	b_first_pos_done:BOOL;
	b_second_pos_done:BOOL;
	b_3rd_pos_done:BOOL;
	b_4th_pos_done:BOOL;
	b_5th_pos_done:BOOL;
	b_6th_pos_done:BOOL;
	b_7th_pos_done:BOOL;
	b_8th_pos_done:BOOL;
	b_9th_pos_done:BOOL;
	b_10th_pos_done:BOOL;
	i_adjust_count:INT:=0;
	adjust_delay:BOOL;
	i_closeloop_count:INT:=0;
	rSPEED: REAL:=2500;
	rACC:REAL:=100;
	rDCC:REAL:=100;
	r_vel_EL_temp:LREAL;
	add_vel:LREAL;
	r_vel_EL:LREAL;
	b_modify_vel: BOOL;
	b_start_adjust_vel:BOOL;
	b_start_adjust_vel_temp:BOOL;
	r_compensation_value_motor: LREAL;
	r_compensation_abs: LREAL;
	b_test_offset_start:BOOL;
	r_offset_az_old:LREAL;
	r_offset_el_old:LREAL;
(*EL  vel mode*)	
	V_LastOutput:LREAL:=0;
	V_LastSpeed:LREAL:=0;
	dIntegralSpeed:LREAL:= 0;	
	V_command_EL:LREAL:=0;
	V_command_EL_V:LREAL:=0;

	V_max_vel_motor:LREAL;
	b_start_cyclicvel: BOOL;
	b_write_el_vel: BOOL;
	m_dLastIntegral:LREAL:=0;
	m_dAUnsub1:LREAL:=0;
	m_dAUnsub2:LREAL:=0;
	m_dAEnsub1:LREAL:=0;
	m_dAEnsub2:LREAL:=0;
	m_dKa:LREAL:=0.5;
	m_dKv:LREAL:=0.1;
	
	speed1:LREAL;
	r_EL_current_when_goto_cmd:LREAL;
	T_count_goto:LREAL;
	Pos_EL_Aim:LREAL;
	r_cyclic_velocity:LREAL;
	r_cyclic_velocity_test:LREAL;
	Pos_EL_error:LREAL;
	b_step_running:BOOL:=0;
	b_step_running_az:BOOL:=0;
	b_step_running_el:BOOL:=0;
	r_step_count:DINT:=0;
	r_step_count_temp:DINT:=0;
	b_offset_running:BOOL;
	r_offset_count_temp:DINT:=0;
	r_offset_count:DINT:=0;
	r_test_offset_az:LREAL;
	r_test_offset_el:LREAL;
	r_Integral_thistime:REAL;
	r_el_offset_abs:LREAL;
END_VAR
VAR_GLOBAL RETAIN PERSISTENT
	AZ_encoder_last: LREAL;
	FI_encoder_last: LREAL;

(*	
	C1:REAL:=-0.504475;
	C2:REAL:=-0.047962;
	C3:REAL:=0.005718;
	C4:REAL:=50.64244;
	C5:REAL:=-0.003995;
	C6:REAL:=0.443004;
	C7:REAL:=0.019635;
	C8:REAL:=0;
*)	

(*	C1:LREAL:=0;
	C2:LREAL:=0;
	C3:LREAL:=0;
	C4:LREAL:=0;
	C5:LREAL:=0;
	C6:LREAL:=0;
	C7:LREAL:=0;
	C8:LREAL:=0;	
*)
	r_pos_motor3_Ini: REAL;

(*	
	P1:LREAL:=0.000000000968559949;
	P2:LREAL:=-0.000000404463748;
	P3:LREAL:=0.0000707747355;
	P4:LREAL:=-0.006745089;
	P5:LREAL:=0.3810258947;
	P6:LREAL:=-13.13945082;
	P7:LREAL:=311.5666046431;
	P8:LREAL:=4122.813236;
	P9:LREAL:=556099.6655657330;
*)
	P1:LREAL:=0.00000000000675664022381225;
	P2:LREAL:=-0.00000000306148315353895;
	P3:LREAL:=0.000000597917575287703;
	P4:LREAL:=-0.0000659096897179393;
	P5:LREAL:=0.00450794567760492;
	P6:LREAL:=-0.198139695223752;
	P7:LREAL:=5.43570049374671;
	P8:LREAL:=-35.3877608207139;
	P9:LREAL:=9702.49448593394;
	P10:LREAL:=422614.297996071;
	
	AA1:LREAL:=0.0000927334099929522;
	AA2:LREAL:=0.0000884282758254779;
	AA3:LREAL:=0.0000846410373605538;
	AA4:LREAL:=0.0000813259380946959;
	AA5:LREAL:=0.0000784067743453034;
	AA6:LREAL:=0.000075826508947528;
	AA7:LREAL:=0.0000735467168745587;
	AA8:LREAL:=0.0000715348517797871;
	AA9:LREAL:=0.0000697632236190369;
	AA10:LREAL:=0.0000682035193015959;
	AA11:LREAL:=0.0000668341977222905;
	AA12:LREAL:=0.0000656452269355495;
	AA13:LREAL:=0.0000646345562191369;
	AA14:LREAL:=0.0000637852732561106;
	AA15:LREAL:=0.000063021502936802;
	
	BB1:LREAL:=37.4712526429021;
	BB2:LREAL:=34.8032470862882;
	BB3:LREAL:=32.2419717976062;
	BB4:LREAL:=29.8041671410679;
	BB5:LREAL:=27.4781245099576;
	BB6:LREAL:=25.2575068243857;
	BB7:LREAL:=23.1452253471404;
	BB8:LREAL:=21.1443430239212;
	BB9:LREAL:=19.2586262226003;
	BB10:LREAL:=17.4866321102168;
	BB11:LREAL:=15.8306154092925;
	BB12:LREAL:=14.3037010778946;
	BB13:LREAL:=12.9288502805138;
	BB14:LREAL:=11.7078506914323;
	BB15:LREAL:=10.5498626131235;
	
END_VAR

// IndraMotionMlc1/Application/UserConstGlobal
VAR_GLOBAL CONSTANT
  // define all possible axis, set to maximum axis index to preserve ressources 
  // set to a maximum of 32 for the L45 and 16? for the L25
  uiMAX_AXIS_INDEX:   UINT    := INT_TO_UINT(MB_MAX_AXIS_NUMBER);
  
  // Simulation related
 	 gc_b_sim_on: BOOL :=0;  // True is simulation code activated. 
  // Azimuth limits
  	gc_r_limit_cw_az_sim:REAL:= 271 ;
	gc_r_limit_ccw_az_sim:REAL:= -271;
	gc_r_limit_final_cw_az_sim:REAL:= 271.2 ;
	gc_r_limit_final_ccw_az_sim:REAL:=-271.2 ;
 // Elevation Limits
	gc_r_limit_cw_el_sim:REAL:= 90.2;
	gc_r_limit_ccw_el_sim:REAL:= 14.8 ;
	gc_r_limit_final_cw_el_sim:REAL:=90.5 ;
	gc_r_limit_final_ccw_el_sim:REAL:=14.5 ;
 // Feed Indexer Limits
	gc_r_limit_cw_fi_sim:REAL:= 108;
	gc_r_limit_ccw_fi_sim:REAL:= -108;
	gc_r_limit_final_cw_fi_sim:REAL:= 108.2 ;
	gc_r_limit_final_ccw_fi_sim:REAL:= -108.2;
  
  // Time related 
  gc_UnixToSKAEpoch: LREAL := 946684768 ; //Seconds
  gc_SKAEpochMJD: LREAL := 51544; // MJD
  gc_KAPB_NTP: STRING :='10.97.64.1';
  gc_ITF_NTP: STRING:= '10.165.3.12 ';
  
 (* // Position limits
  gc_r_pos_max_Az: REAL := 271;
  gc_r_pos_min_Az: REAL := -271;  
  gc_r_pos_max_El: REAL := 90.2;
  gc_r_pos_min_El: REAL := 14.8;  
  gc_r_pos_max_Fi: REAL := 106;
  gc_r_pos_min_Fi: REAL := -106;  *)

   // Position limits
  gc_r_pos_max_Az: REAL := 271;
  gc_r_pos_min_Az: REAL := -271;  
  gc_r_pos_max_El: REAL := 90.20;
  gc_r_pos_min_El: REAL := -14.80;  
  gc_r_pos_max_Fi: REAL := 106;
  gc_r_pos_min_Fi: REAL := -106;  
  
  
  // Velocity limits
   gc_r_vel_max_Az: REAL := 0.5; //3/6; //scaling RPM of Axis  Deg/s = 6* RPM 
   gc_r_vel_max_El: REAL := 0.16667;
   gc_r_vel_max_Fi: REAL := 2;
   
  // Power limiting
     gc_r_power_Kv_Az: REAL := 0.05;//0.3Deg/s/kW;
  	 gc_r_power_Kv_El: REAL := 0.016667;// 0.1;
     gc_r_power_Kv_Fi: REAL := 0.2;//1.2;
	 gc_r_power_Ka_Az: REAL := 0.055;
  	 gc_r_power_Ka_El: REAL := 0.002;
  	 gc_r_power_Ka_Fi: REAL := 0.1; 

     
   // Tracking  If the velocity is below this limit then then the dish is tracking abovethe limit it is slewing. 
   gc_r_vel_tracking_limit_Az: REAL := 1;  // Scaling
   gc_r_vel_tracking_limit_El: REAL := 0.4;
   gc_r_vel_tracking_limit_Fi: REAL := 0;
   
   // Stop Deceleration values  
  gc_r_Stop_dec_Az: REAL := 0.5; //Rad/s^2
  gc_r_Stop_dec_El: REAL := 0.5; // 28,64 deg/s^2
  gc_r_Stop_dec_Fi: REAL := 0.5;
  
   // Stop Deceleration values  
  gc_r_limit_Stop_dec_Az: REAL := 5; //Rad/s^2
  gc_r_limit_Stop_dec_El: REAL := 5; // 28,64 deg/s^2
  gc_r_limit_Stop_dec_Fi: REAL := 5;
  
  
  // Goto Acceleration Values
  gc_r_goto_acc_Az: REAL := 0.02; //Rad/s^2 
  gc_r_goto_acc_El: REAL := 0.02; // 1.14 deg/s^@
  gc_r_goto_acc_Fi: REAL := 0.2; // 11.4 deg/s^2
  
  // Feed indexer positions for bands
  gc_r_band_tolerance: REAL := 0.001; // Tolerance for being in position
  gc_r_band_optical : REAL := 0;
  gc_r_band_1 : REAL := 103.37;
  gc_r_band_2 : REAL := -99.97;
  gc_r_band_3 : REAL := -47.684;
  gc_r_band_4 : REAL := 10.444;
  gc_r_band_5a : REAL := -6.398;
  gc_r_band_5b : REAL := -30.842;
  gc_r_band_6 : REAL := -18.62;
  
  // Stow Positions
  gc_r_stow_Az: REAL :=0; 
  gc_r_stow_El: REAL :=90;
  gc_stow_horn_alarm_time: TIME := T#5S;
  gc_UPS_Stow_Az_Speed: REAL := 0.16667;
  gc_UPS_Stow_El_Speed: REAL := 0.083; 
  // AutoStow 
  gc_i_autostow_counter_max: INT := 2; 
  
  // Static off set limits
  gc_r_Xel_off_limit: REAL := 36000; // arcsec
  gc_r_El_off_limit: REAL := 36000;
	 
  // Pointing 
  gc_stack_length: INT :=10000; 
  gc_r_tilt_vel_limit_Az: REAL := 1; // deg/s	 
  gc_lr_tilt_corr_limit_Az: LREAL:= 1000; //arcseconds 
  gc_lr_tilt_corr_limit_El: LREAL:= 1000; //arcseconds 
  gc_lr_arcsec2deg: LREAL:=3600;
  gc_lr_point_corr_error_lim : LREAL := 360000; //arcseconds
  
  // DAM 
  gc_st_DAM_ip:String :='192.168.1.222';
	 
END_VAR

// IndraMotionMlc1/Application/UserVarGlobal
VAR_GLOBAL 
  // Axis interface: command structure: define as RETAIN, to keep the values 
  // Note: on the L40.2 control, the RETAIN memory is slower then normal VAR, so define 
  //       this structure only as RETAIN when necessary 
  //  arAxisCtrl_gb: ARRAY [1..MAX_AXIS_NUM] OF MB_AXIS_CONTROL;
	
  // Axis interface: command structure 
  arAxisCtrl_gb: ARRAY [1..uiMAX_AXIS_INDEX] OF TE_AXIS_CONTROL_TYPE01;
END_VAR

VAR_GLOBAL
//----------------------------------- Machine status variables ----------------------------	

  // Axis interface: status structure 
  arAxisStatus_gb: ARRAY [1..uiMAX_AXIS_INDEX] OF TE_AXIS_STATUS_TYPE01;

  bRemoteOn_gb  : BOOL := FALSE;  // TRUE: Internal IL visu is active 
                                  // FALSE: PlcProg is active

  
END_VAR

// IndraMotionMlc1/Application/AxisInterface/Global_AxIf_Const
{attribute 'qualified_only'}
VAR_GLOBAL CONSTANT
    // define masks for the sync operating modes 
    // e.g. IF( (INT_TO_WORD(AdminStatus._OpMode.enAck) AND MASK_MODE_WITH_FINE_ADJ) <> 0 ) THEN 
    MASK_MODE_PHASE_SHIFT   :DWORD := 16#0BC0; (* SYNC_PHASE, SYNC_CAM, SYNC_PROFILE, FLEX_PROFILE, SYNC_VEL *)
END_VAR
VAR_GLOBAL

END_VAR

// IndraMotionMlc1/Application/AxisInterface/Global_Axis_Interface
{attribute 'linkalways'}
{attribute 'analysis' := '-33'} // disable static code analysis rule 33, check of unused variable
VAR_GLOBAL
    (* Axis number for the visualization screens *)
    VisuAxisNo : INT := 1;
    
	  arAxisIdx_gb: ARRAY [1..uiMAX_AXIS_INDEX] OF UINT; // list of all axes index without gaps 
    uiNofAxis_gb: UINT; // number of axis in C-0-0484
    
END_VAR

// IndraMotionMlc1/Application/PLC_PRG
VAR_GLOBAL
		
Safety:fb_Safety;
CommandArbiter:fb_CommandArbiter;
Time_cds:fb_Time_cds;
Pointing:fb_Pointing;
Tracking:fb_Tracking;
Management:fb_Management;
Azimuth:fb_Axis;
Elevation:fb_Axis;
FeedIndexer:fb_Axis;





	
(************CommandArbiter ************)	

	Authority:STRING:='LMC';    (* the authority for DSC control now*)
	Command_Arbiter_error:BOOL;(*Command Arbiter error*)

(****************Management*******************)

	DsState:UINT;(*The Dish state 0Startup 1Standby 2Locked 3Estop 4Stowed 5Lcok&Stowed 6Activating 7Deactivating 8Standstill 9Stop 10Slew 11jog 12Track*)
	Current_FIPos:UINT;(*Current position of the FI*)
	r_operation_hour: LREAL;(*FP_C_0_0051,Operation hour counter*)
	K_gear_ratio:LREAL:=1800;// The ratio beteen the leadscrew length and elevation angle This variable needs a non-zero startup to prevent divide by zero.
	HumidDriveCab: LREAL;
	HumidDriveCab_Up: LREAL;
	HumidPSC_Inlet: LREAL;
	HumidPSC_Outlet: LREAL;
	TempDriveCab: LREAL;
	TempDriveCab_Up: LREAL;
	TempEMISC_Outlet: LREAL;
	TempPSC_Inlet: LREAL;
	TempPSC_Outlet: LREAL;
	CurrentPh1: LREAL;
	CurrentPh2: LREAL;
	CurrentPh3: LREAL;
	FrequencyPh1: LREAL;
	FrequencyPh2: LREAL;
	FrequencyPh3: LREAL;
	PowerFactor: LREAL;
	VoltagePh1: LREAL;
	VoltagePh2: LREAL;
	VoltagePh3: LREAL;
	
	Pedestal_temp_1: REAL;
	Pedestal_temp_2 : REAL;
	Pedestal_temp_3 : REAL;
	
	ActivePowerConsumption: LREAL;
	ReactivePowerConsumption: LREAL;
	ApparentPowerConsumption: LREAL;
		
(********************Time**********************)	
	Source_Timesync:UINT:=2;(*Time source, 0 PTP 1 NTP 2 DSC*)
	IP_Adress_PTP:STRING;(* The PTP server adresss*)
	IP_Adress_NTP:STRING;(* The PTP server adresss*)
	//DscTime:DATE_AND_TIME;(*DSC internal time*)
	//TimeSynced:BOOL;(*The time is synced to the source*)
	
(**********************Pointing************************)	
	(*ActAmbTemp_East:LREAL;
	ActAmbTemp_South:LREAL;
	AmbTempCorrVal_1:LREAL;
	AmbTempCorrVal_2:LREAL;
	TiltXRaw_One:LREAL;
	TiltYRaw_One:LREAL;
	TiltXArcsec_One:LREAL;
	TiltYArcsec_One: BOOL;
	TiltXFilt_One:LREAL;
	TiltYFilt_One:LREAL;
	TiltTemp_One:LREAL;
	TiltXRaw_Two:LREAL;
	TiltYRaw_Two:LREAL;
	TiltXArcsec_Two:LREAL;
	TiltYArcsec_Two: BOOL;
	TiltXFilt_Two:LREAL;
	TiltYFilt_Two:LREAL;
	TiltTemp_Two:LREAL;
	TiltCorrVal_Az:LREAL;
	TiltCorrVal_EL:LREAL;
	PmCorrVal_Az: BOOL;
	PmCorrVal_EL: BOOL;
	StaticCorrActive:BOOL;
	TiltCorrActive:BOOL;
	Pointing_TiltOn:UINT;
	TempCorrActive:BOOL;
	BandForCorr:UINT;*)
	Pointing_TiltOn:UINT;
(**************************Tracking********************************)
(*	tr_initOk:BOOL;(*Tracking function program is initialized and ready for operation*)
	tr_valid:BOOL;(*The tracking controller’s output is within the position ranges of the dish structure.*)
	tr_Table_error:BOOL;(*The table reports an error *)
	tr_obj_valid:BOOL;(*Tracking object has valid tracking data.*)
	tr_selFIy:BOOL;(*FIynomial tracking selected as source*)
	act_statOffset_value_Xel:LREAL;(*Actual azimuth static offset*)
	act_statOffset_value_El:LREAL;(*Elevation azimuth static offset*)
	p_desired_AZ:LREAL;(*Azimuth position output of the Tracking Controller*)
	p_desired_EL:LREAL;(*Elevation position output of the Tracking Controller*)
	tr_TimeRemaining:LREAL;(*Time till the last point in the track table is reached*)
	OnSourceDev:LREAL;(*Actual calculated “On Sky” rms tracking error.*) *)
(*********Read parameteers*******)
	AxRef:ARRAY[1..5] OF AXIS_REF;
	P_shape_value:ARRAY[1..5] OF LREAL;
	V_shape_value:ARRAY[1..5] OF LREAL;
	V_act_value:ARRAY[1..5] OF LREAL;
	r_write_position_az: LREAL; // Used internally for interpolator and pointing model calculations
    r_write_position_az_out: LREAL; (*the position written to the virvual azimuth axis*)
	r_write_position_el: LREAL; // Used internally for interpolator and pointing model calculations
    r_write_position_el_out: LREAL;(*the position written to the virvual elevation axis*)
	r_write_position_FI: LREAL;(*the position written to the virvual FeedIndexer axis*)
	r_write_position_FI_out: LREAL;(*the position written to the virvual FeedIndexer axis*)
	
END_VAR

VAR_GLOBAL RETAIN PERSISTENT
	R_total_distance_AZ:LREAL;
	R_total_distance_EL_deg:LREAL;
	R_total_distance_EL_m:LREAL;
	R_total_distance_FI:LREAL;
	
	LeapSecPTP: UINT :=37;    // Storage for Leap seconds 
	
END_VAR

// IndraMotionMlc1/Application/POUs/Motion/P_Position_and_MJD
(*The program is built for calculating the position of real axis, virtual axis and the MJD time,
and writing software limit of azimuth *)
PROGRAM P_Position_and_MJD
VAR
(*With the function block "MB_WriteRealParameter" you can write a defined value to the parameter belonging to the parameter number*)
	fb_write_negative_a: MB_WriteRealParameter;
	fb_write_negative_s: MB_WriteRealParameter;
	fb_write_positive_a: MB_WriteRealParameter;
	fb_write_positive_s: MB_WriteRealParameter;
(*the blink function block is for triggering MB_WriteRealParameter function block*)
	fb_blink_1: BLINK;
	fb_blink_2: BLINK;
	fb_blink_3: BLINK;
	fb_blink_4: BLINK;
(*the value is written to MB_WriteRealParameter*)
	r_negative_limit: REAL;
	r_positive_limit: REAL;
(*the elevation limit control*)
	fb_blink_diagnos_el: BLINK;
	fb_diagnose_el: MB_ReadStringParameter;
	str_diagnose_el: STRING;
	fb_blink_5: BLINK;
	fb_blink_6: BLINK;
	fb_write_negative_el: MB_WriteRealParameter;
	fb_write_positive_el: MB_WriteRealParameter;
	r_limit_el_up: REAL;
	r_limit_el_down: REAL;
	b_limit_up_el: BOOL;
	b_limit_down_el: BOOL;
	rtrig_set_limit_up: R_TRIG;
	rtrig_set_limit_down: R_TRIG;
	fb_blink_7: BLINK;
	fb_write_91_az1: MB_WriteRealParameter;
	fb_blink_8: BLINK;
	fb_blink_9: BLINK;
	fb_blink_10: BLINK;
	fb_blink_11: BLINK;
	fb_write_91_az2: MB_WriteRealParameter;
	fb_write_91_el1: MB_WriteRealParameter;
	fb_write_91_el2: MB_WriteRealParameter;
	fb_write_91_FI: MB_WriteRealParameter;
	fb_blink_12: BLINK;
	fb_write_91_FI2: MB_WriteRealParameter;
	r_pos_FI_1: REAL;
	i_counter_hr: BOOL;
	rtrig_hr:R_TRIG;
	
	fb_blink_111: BLINK;
	fb_write_negative_a_v: MB_WriteRealParameter;
	fb_blink_1_v: BLINK;
	fb_blink_2_v: BLINK;
	fb_write_negative_s_v: MB_WriteRealParameter;
	fb_blink_3_v: BLINK;
	fb_write_positive_a_v: MB_WriteRealParameter;
	
	temp_a:LREAL:=3135.4451;
	temp_b:LREAL:=3013.785;	
	temp_c:LREAL;
	r_pos_az_org :LREAL;
	r_pos_az_v_org :LREAL;
	r_pos_el_org:LREAL;
	r_pos_el_v_org:LREAL;

	fb_real_drive3_s51: MB_ReadRealParameter;
	r_pos_motor3_1: REAL;
	
	i_overlop:BOOL;
	rtrig_overlop:R_TRIG;
	
	
	DeltaB_temp: LREAL;
	
	B_TEMP: LREAL;
	
	MB_AxisDistanceAccumulator_2: MB_AxisDistanceAccumulator;
	bDisenable1: BOOL;
	test_1: LREAL;
	test_2: LREAL;
	test_old: LREAL;
	normal_count:DINT:=995;
	low_count:DINT:=9995;
	fast_count:DINT:=9995;
	i_change_sign_count:DINT;
	r_threshold:REAL;
END_VAR
VAR RETAIN
	r_last_position_az: REAL:=1;
	l_control:LREAL;
	a_control:REAL:=3035.4;
	b_control:REAL:=3035.1;
	b_motor_count:DINT:=0;
	b_sign_delay:BOOL:=0;
	b_sign_delay_count:DINT:=0;
	r_test_value:LREAL;
	i_test_value:DINT:=0;
	fb_read_source_code_3: MB_ReadParameter;
	r_source_code_3: DINT;
	r_source_to_elevation: LREAL;
END_VAR

 	//axisdata[7].rActualPosition_i;
r_source_to_elevation:=(DINT_TO_LREAL(r_source_code_3)/536870912)*360.0-64.812477;

	MB_AxisDistanceAccumulator_2(
	Enable:= bDisenable1, 
	TotalDistance:= 1000000, 
	InOperation=> , 
	Error=> , 
	ErrorID=> , 
	ErrorIdent=> , 
	DistanceReached=> , 
	AccumulatedDistance=> r_length_Distance_1, 
	Axis:= Drive3);
	
	IF	r_pos_motor3<0.01 AND r_pos_motor3>=0 THEN
	i_overlop:=TRUE;
	ELSE
	i_overlop:=FALSE;
	END_IF	
	rtrig_overlop(clk:=i_overlop);
	IF rtrig_overlop.Q=TRUE THEN
	b_motor_count:=b_motor_count+1;
	END_IF
		
	l_control:=SQRT(a_control*a_control+b_control*b_control-2*a_control*b_control*COS(deg2rad(112.0255-ML_Base.AxisData[3].rActualPosition_i)))-1151;
//	
//	temp_c:= SQRT(temp_a*temp_a + temp_b*temp_b-2*temp_a*temp_b*COS((115.5-r_pos_el_v)*3.1415926/180.0));
//	gear_ratio:=temp_a*temp_b*SIN((115.5-r_pos_el_v)*3.1415926/180.0)/temp_c*6.0*168.0/25.0/180.0*3.1415926;
	
	

(*<<time1<<<<<<<<<<<<<<<<<<<<<<<<<<<<<< real position of azimuth elevation and FeedIndexer>>>>>>>>>>>>>>>>>>>>>>>>>>>>>>>>*)
(*the azimuth position is judged by zone signal*)

	IF axisdata[1].Axis_Inbb=TRUE THEN	
		//r_pos_az_org:=axisdata[1].rActualPosition_i;
		//r_pos_az_1:=r_pos_az_org+C1+C3*SIN((r_pos_az_org-C4)*3.1415926/180)*TAN(r_pos_el_org*3.1415926/180)+C5*TAN(r_pos_el_org*3.1415926/180)+C6/COS(r_pos_el_org*3.1415926/180);		
	//	r_pos_az_modify:=r_pos_az_1;
	    r_pos_az_modify:=axisdata[1].rActualPosition_i;
		IF r_pos_az_1>=360.0 THEN 
			r_pos_az_modify:=r_pos_az_1-360.00;
		END_IF
		IF r_pos_az_1<0.0 THEN 
			r_pos_az_modify:=r_pos_az_1+360.00;
		END_IF
			
	END_IF;		
	
  (* IF gc_b_sim_on THEN
	   IF b_zone_az_sim=FALSE THEN
			r_pos_az:=axisdata[1].rActualPosition_i-360;
			r_pos_az_v:=axisdata[7].rActualPosition_i-360;
        ELSE
       r_pos_az:=axisdata[1].rActualPosition_i;
		r_pos_az_v:=axisdata[7].rActualPosition_i;
		END_IF;
	IF ABS (r_pos_az_v ) = 360 THEN	
	 //r_pos_az:=0.0000;
	// r_pos_az_v := 0.0000;
	 END_IF
   ELSE 
	 r_pos_az:=axisdata[1].rActualPosition_i;
	 r_pos_az_v:=axisdata[7].rActualPosition_i;
   END_IF*)
   IF b_zone_az=FALSE AND axisdata[1].rActualPosition_i>75 AND axisdata[1].rActualPosition_i<360 THEN
			r_pos_az:=axisdata[1].rActualPosition_i-360;
			r_pos_az_v:=axisdata[1].rActualPosition_i-360;
//		ELSIF axisdata[1].rActualPosition_i>299 THEN
	//		r_pos_az:=axisdata[1].rActualPosition_i-360;
//			r_pos_az_v:=axisdata[1].rActualPosition_i-360;
        ELSE
        r_pos_az:=axisdata[1].rActualPosition_i;
		r_pos_az_v:=axisdata[1].rActualPosition_i;
		END_IF;
//	r_pos_az:=axisdata[1].rActualPosition_i;
//	r_pos_az_v:=axisdata[1].rActualPosition_i;
	AZ_encoder_last:=r_pos_az_v;
	
	IF axisdata[5].rActualPosition_i < 180 THEN
		r_pos_Fi:=axisdata[5].rActualPosition_i;
	    r_pos_Fi_v:=axisdata[5].rActualPosition_i;
	ELSE
		r_pos_Fi:=axisdata[5].rActualPosition_i-360;
	    r_pos_Fi_v:=axisdata[5].rActualPosition_i-360;
		//angleerror := axisdata[1].rActualPosition_i - axisdata[2].rActualPosition_i;
	END_IF
	FI_encoder_last:=r_pos_fi_v;
	
//r_pos_el_org:=axisdata[3].rActualPosition_i;
//r_pos_el_1:=r_pos_el_org+C2+C3*COS((r_pos_az_org-C4)*3.1415926/180)+C7*COS(r_pos_el_org*3.1415926/180)+0;	
//r_pos_el_modify	:=r_pos_el_1;
//r_pos_el:=axisdata[3].rActualPosition_i;
//r_pos_el:=r_source_to_elevation;
//r_pos_el_v:=axisdata[3].rActualPosition_i;

r_pos_el:=ML_Base.AxisData[11].rActualPosition_i;
r_pos_el_v:=ML_Base.AxisData[11].rActualPosition_i; 

(*<<<<<<<<<<<<<<<<<<<<<<<<<<<<<<<<<<<<<<<<<<<<<<<<<<<calculation for MJD >>>>>>>>>>>>>>>>>>>>>>>>>>>>>>>>>>>>>>>*)
(*the definition of MJD is shown in the global variables*)
(*the module of v_time_master axis is 360,so that it take 6minuts to run one cycle*)
IF	axisdata[10].rActualPosition_i<0.01 AND axisdata[10].rActualPosition_i>=0 THEN
	i_counter_hr:=TRUE;
ELSE
	i_counter_hr:=FALSE;
END_IF	
rtrig_hr(clk:=i_counter_hr);
IF rtrig_hr.Q=TRUE THEN
	i_num_quarter:=i_num_quarter+1;
END_IF
IF i_num_quarter=240 THEN
	i_num_quarter:=0;
	di_MJD_day:=di_MJD_day+1;
END_IF

//lr_MJD_current:=TO_REAL(di_MJD_day)+(360*TO_REAL(i_num_quarter)+axisdata[10].rActualPosition_i)/86400+1.0/3.0; // Sets MJD to Beijing time
lr_MJD_current:=TO_REAL(di_MJD_day)+(360*TO_REAL(i_num_quarter)+axisdata[10].rActualPosition_i)/86400;
lr_TAIoffset_current:= (lr_MJD_Current-gc_SKAEpochMJD)*86400+(time_cds.Status.LeapSecPTP); // Minus 10s if you want to correlate to a unix timestamp


(*<<<<<<<<<<<<<<<<<calculate the following error of trajectory>>>>>>>>>>>>>>>>>>>*)

IF ABS(r_vel_EL)>=0.5 THEN
	r_threshold:=0.25;
ELSE 
	r_threshold:=0.15;
END_IF

IF b_open_channel_az AND b_open_channel_el THEN
//IF ABS(lr_MJD_current-track_table[i_start].MJD-0.0000000254)*86400<=0.0005 AND b_sign_delay=0 THEN
	IF ABS(lr_TAIoffset_current-track_table[i_start].TAIoffset-0.0022)<=0.0005 AND b_sign_delay=0 THEN
	b_sign_delay:=1;
//	r_test_value:=0;
	i_test_value:=0;
	r_track_error[1]:=track_table[i_start].Azimuth-r_pos_az;
	
(*   For Elevation orientation axis

	r_track_error[2]:=track_table[i_start].Elevation_ori+r_offset_el_program-r_pos_el;
   IF ABS(r_track_error[2])<r_threshold THEN
		test_1:=Encoder_to_motor(track_table[i_start].Elevation_ori)-Encoder_to_motor(track_table[i_start].Elevation_ori-r_track_error[2]);
		test_2:=Encoder_to_motor(track_table[i_start].Elevation_ori)-Encoder_to_motor(track_table[i_start].Elevation_ori+r_track_error[2]);
//		test_3:=test_1+test_old;
	ELSE
		test_1:=0;
		test_2:=0;
		r_compensation_abs:=0;
		test_old:=0;
	END_IF *)
	
END_IF
	IF b_sign_delay =1 THEN

	i_test_value:=i_test_value+1;
	
	IF i_test_value>995 THEN 
		r_test_value:=r_compensation_abs;
	ELSE
		r_test_value:=r_compensation_abs+test_1/995;
	END_IF
		r_compensation_abs:=r_test_value;
		
	END_IF
		
	END_IF

IF b_sign_delay =1 THEN 
	b_sign_delay_count:=b_sign_delay_count+1;
END_IF

IF ABS(r_vel_EL)<0.002 THEN
	i_change_sign_count:=9995;
ELSIF ABS(r_vel_EL)>0.6 AND ABS(r_vel_EL)<0.8 THEN
	i_change_sign_count:=9995;
ELSIF ABS(r_vel_EL)>=0.8 THEN
	i_change_sign_count:=12995;	
ELSE 
	i_change_sign_count:=normal_count;	
END_IF


IF b_sign_delay_count>i_change_sign_count THEN
	b_sign_delay_count:=0;
	b_sign_delay:=0;
END_IF


IF b_off_write=TRUE THEN
	r_limit_s91:=11;
ELSE
	r_limit_s91:=1.4;
END_IF;
(*<<<<<<<<<<<<<<<<<<the azimuth limit control>>>>>>>>>>>>>>>>>>>>*)
IF (r_pos_az<-250) OR (r_pos_az>250) THEN
(*the range of azimuth is -179~359*)
	//r_negative_limit:=89;
	//r_positive_limit:=271;
	r_negative_limit:=gc_r_limit_ccw_az_sim;
	r_positive_limit:=gc_r_limit_cw_az_sim;
ELSE
	//r_negative_limit:=0;
	//r_positive_limit:=360;
	r_negative_limit:=gc_r_limit_ccw_az_sim;
	r_positive_limit:=gc_r_limit_cw_az_sim;
END_IF;
(*
(*<<<<<<<<<<<<<<<<<<<<<<<<<the elevation limit control>>>>>>>>>>>>>>>>>>>>>>>*)
IF str_diagnose_el='F6029 ' THEN
	b_limit_up_el:=TRUE;
ELSE
	b_limit_up_el:=FALSE;
END_IF
rtrig_set_limit_up(clk:=b_limit_up_el);
IF rtrig_set_limit_up.Q=TRUE THEN
	r_limit_el_up:=90.05;
END_IF
IF r_pos_el <=90.1 THEN
	r_limit_el_up:=90.15;
END_IF

IF str_diagnose_el='F6030 ' THEN
	b_limit_down_el:=TRUE;
ELSE
	b_limit_down_el:=FALSE;
END_IF
rtrig_set_limit_down(clk:=b_limit_down_el);
IF rtrig_set_limit_down.Q=TRUE THEN
	r_limit_el_down:=14.7;
END_IF
IF r_pos_el >=14.65 THEN
	r_limit_el_down:=14.6;
END_IF
*)



//P_Position_and_MJD.A_Write_Limit_Value();lr_TAIoffset_current
//Time Sensitive pointing data
Time_cds.Status.TAIOffset:=lr_TAIoffset_current;
(*IF gc_b_sim_on THEN 
	IF r_pos_az = -360 THEN
		r_pos_az:= 0;
	END_IF

END_IF
*)
Azimuth.Status.p_Act:=pointing.Status.TotalPointCorr_Az/gc_lr_arcsec2deg+r_pos_az;
Azimuth.Status.p_Enc:=r_pos_az;
Elevation.Status.p_Act:=pointing.Status.TotalPointCorr_El/gc_lr_arcsec2deg+r_pos_el;
Elevation.Status.p_Enc:=r_pos_el;

Pointing.Status.CurrentPointing[0]:= Time_cds.Status.TAIoffset;
Pointing.Status.CurrentPointing[1]:= Azimuth.Status.p_Act;
Pointing.Status.CurrentPointing[2]:= Elevation.Status.p_Act;
Pointing.Status.CurrentPointing[3]:= Azimuth.Status.p_Enc;
Pointing.Status.CurrentPointing[4]:= Elevation.Status.p_Enc;
Pointing.Status.CurrentPointing[5]:= pointing.Status.TiltCorrVal_Az;
Pointing.Status.CurrentPointing[6]:= pointing.Status.TiltCorrVal_El;

ACTION A_Write_Limit_Value:
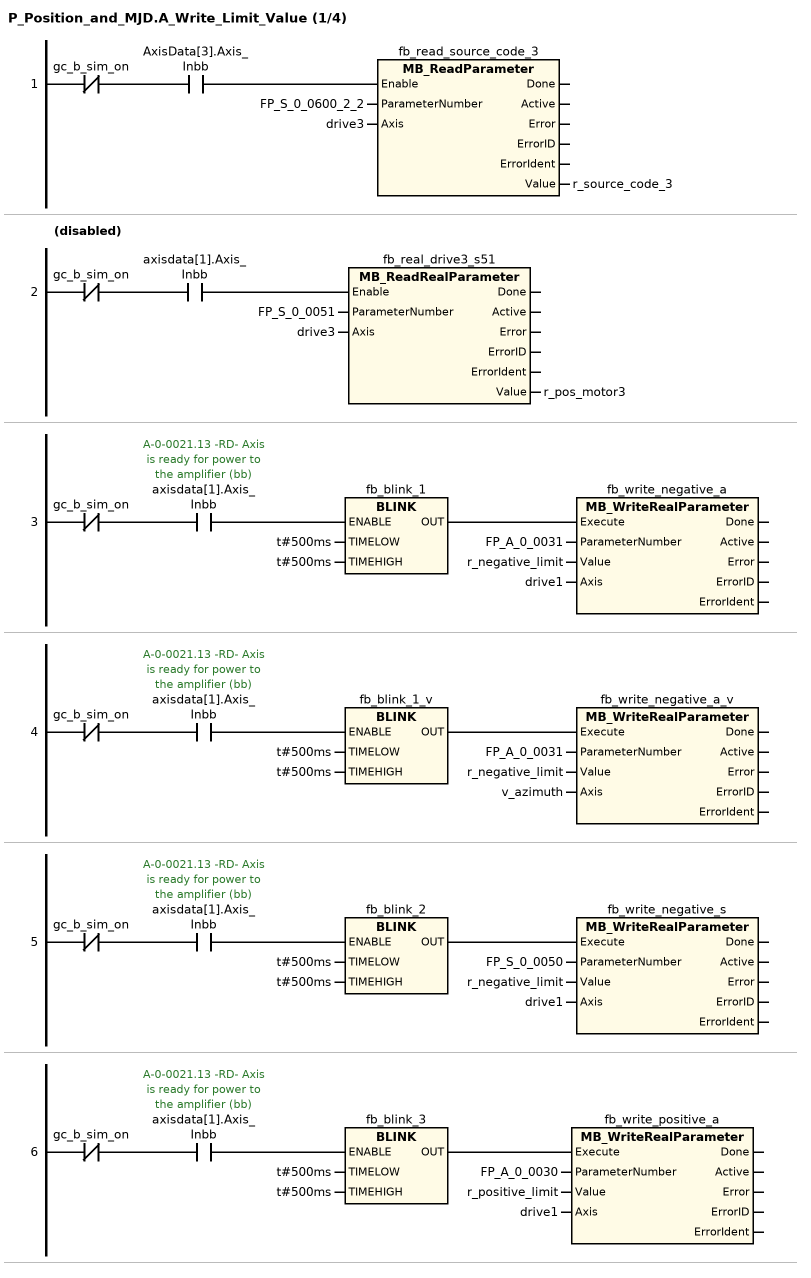
// NETWORK 1
fb_read_source_code_3(
    Enable := NOT gc_b_sim_on AND AxisData[3].Axis_Inbb,
    ParameterNumber := FP_S_0_0600_2_2,
    Axis := drive3,
    Value => r_source_code_3); // MB_ReadParameter

// NETWORK 2 (disabled)
//   FP_S_0_0051: Position limit value, negative
//   drive3: the value is written to MB_WriteRealParameter
// fb_real_drive3_s51(
//     Enable := NOT gc_b_sim_on AND axisdata[1].Axis_Inbb,
//     ParameterNumber := FP_S_0_0051,
//     Axis := drive3,
//     Value => r_pos_motor3); // MB_ReadRealParameter

// NETWORK 3
//   fb_write_negative_a: With the function block "MB_WriteRealParameter" you can write a defined value to the parameter belonging to the parameter number
//   fb_blink_1: the blink function block is for triggering MB_WriteRealParameter function block
//   axisdata[1].Axis_Inbb: A-0-0021.13 -RD- Axis is ready for power to the amplifier (bb)
//   FP_A_0_0031: Position limit value, negative
//   r_negative_limit: the value is written to MB_WriteRealParameter
//   drive1: Real axis "Drive1" with axis number 1
fb_blink_1(ENABLE := NOT gc_b_sim_on AND axisdata[1].Axis_Inbb, TIMELOW := t#500ms, TIMEHIGH := t#500ms); // BLINK
fb_write_negative_a(
    Execute := fb_blink_1.OUT,
    ParameterNumber := FP_A_0_0031,
    Value := r_negative_limit,
    Axis := drive1); // MB_WriteRealParameter

// NETWORK 4
//   axisdata[1].Axis_Inbb: A-0-0021.13 -RD- Axis is ready for power to the amplifier (bb)
//   FP_A_0_0031: Position limit value, negative
//   r_negative_limit: the value is written to MB_WriteRealParameter
//   v_azimuth: Virtual axis "v_azimuth" with axis number 7
fb_blink_1_v(ENABLE := NOT gc_b_sim_on AND axisdata[1].Axis_Inbb, TIMELOW := t#500ms, TIMEHIGH := t#500ms); // BLINK
fb_write_negative_a_v(
    Execute := fb_blink_1_v.OUT,
    ParameterNumber := FP_A_0_0031,
    Value := r_negative_limit,
    Axis := v_azimuth); // MB_WriteRealParameter

// NETWORK 5
//   axisdata[1].Axis_Inbb: A-0-0021.13 -RD- Axis is ready for power to the amplifier (bb)
//   FP_S_0_0050: Negative position limit value
//   r_negative_limit: the value is written to MB_WriteRealParameter
//   drive1: Real axis "Drive1" with axis number 1
fb_blink_2(ENABLE := NOT gc_b_sim_on AND axisdata[1].Axis_Inbb, TIMELOW := t#500ms, TIMEHIGH := t#500ms); // BLINK
fb_write_negative_s(
    Execute := fb_blink_2.OUT,
    ParameterNumber := FP_S_0_0050,
    Value := r_negative_limit,
    Axis := drive1); // MB_WriteRealParameter

// NETWORK 6
//   axisdata[1].Axis_Inbb: A-0-0021.13 -RD- Axis is ready for power to the amplifier (bb)
//   FP_A_0_0030: Position limit value, positive
//   drive1: Real axis "Drive1" with axis number 1
fb_blink_3(ENABLE := NOT gc_b_sim_on AND axisdata[1].Axis_Inbb, TIMELOW := t#500ms, TIMEHIGH := t#500ms); // BLINK
fb_write_positive_a(
    Execute := fb_blink_3.OUT,
    ParameterNumber := FP_A_0_0030,
    Value := r_positive_limit,
    Axis := drive1); // MB_WriteRealParameter

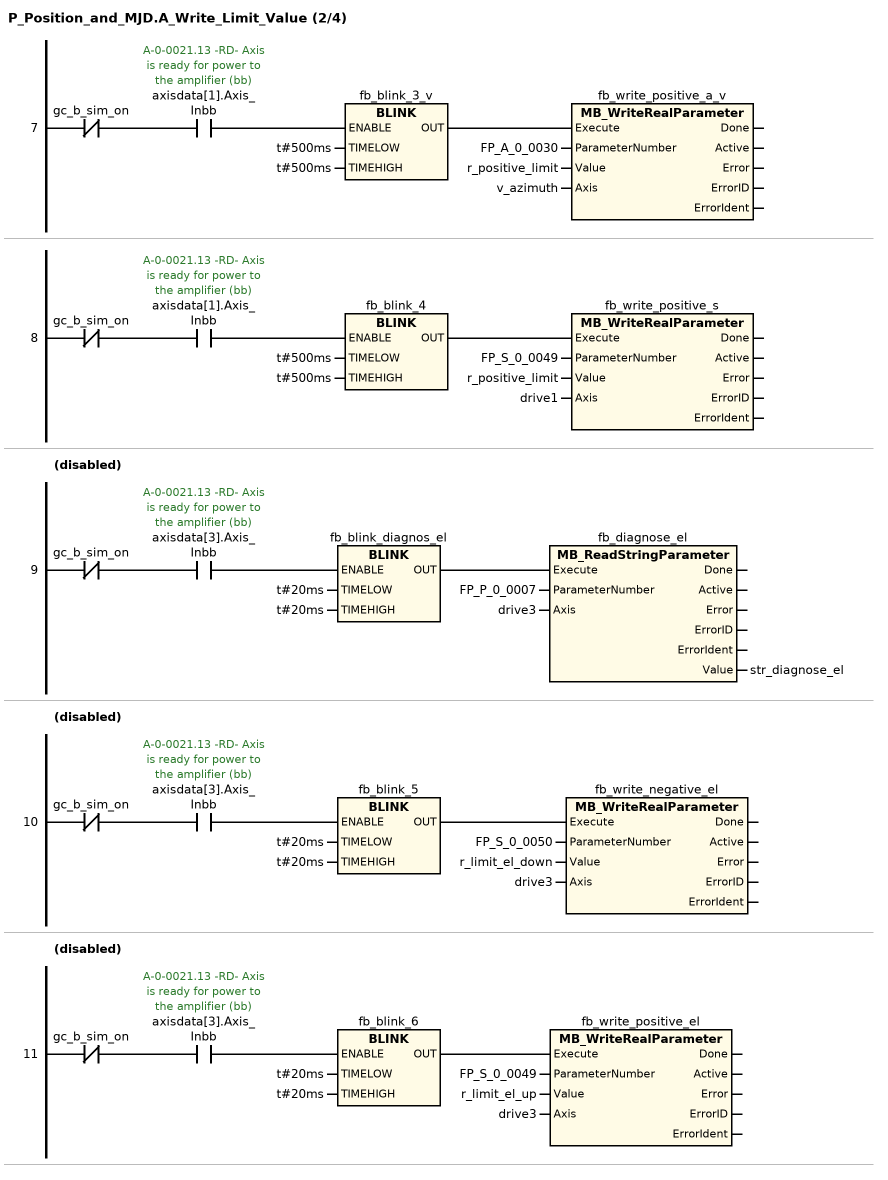
// NETWORK 7
//   axisdata[1].Axis_Inbb: A-0-0021.13 -RD- Axis is ready for power to the amplifier (bb)
//   FP_A_0_0030: Position limit value, positive
//   v_azimuth: Virtual axis "v_azimuth" with axis number 7
fb_blink_3_v(ENABLE := NOT gc_b_sim_on AND axisdata[1].Axis_Inbb, TIMELOW := t#500ms, TIMEHIGH := t#500ms); // BLINK
fb_write_positive_a_v(
    Execute := fb_blink_3_v.OUT,
    ParameterNumber := FP_A_0_0030,
    Value := r_positive_limit,
    Axis := v_azimuth); // MB_WriteRealParameter

// NETWORK 8
//   axisdata[1].Axis_Inbb: A-0-0021.13 -RD- Axis is ready for power to the amplifier (bb)
//   FP_S_0_0049: Positive position limit value
//   drive1: Real axis "Drive1" with axis number 1
fb_blink_4(ENABLE := NOT gc_b_sim_on AND axisdata[1].Axis_Inbb, TIMELOW := t#500ms, TIMEHIGH := t#500ms); // BLINK
fb_write_positive_s(
    Execute := fb_blink_4.OUT,
    ParameterNumber := FP_S_0_0049,
    Value := r_positive_limit,
    Axis := drive1); // MB_WriteRealParameter

// NETWORK 9 (disabled)
//   fb_blink_diagnos_el: the elevation limit control
//   axisdata[3].Axis_Inbb: A-0-0021.13 -RD- Axis is ready for power to the amplifier (bb)
//   FP_P_0_0007: Display text of diagnostic message
//   drive3: Real axis "Drive3" with axis number 3
// fb_blink_diagnos_el(
//     ENABLE := NOT gc_b_sim_on AND axisdata[3].Axis_Inbb,
//     TIMELOW := t#20ms,
//     TIMEHIGH := t#20ms); // BLINK
// fb_diagnose_el(
//     Execute := fb_blink_diagnos_el.OUT,
//     ParameterNumber := FP_P_0_0007,
//     Axis := drive3,
//     Value => str_diagnose_el); // MB_ReadStringParameter

// NETWORK 10 (disabled)
//   axisdata[3].Axis_Inbb: A-0-0021.13 -RD- Axis is ready for power to the amplifier (bb)
//   FP_S_0_0050: Negative position limit value
//   drive3: Real axis "Drive3" with axis number 3
// fb_blink_5(ENABLE := NOT gc_b_sim_on AND axisdata[3].Axis_Inbb, TIMELOW := t#20ms, TIMEHIGH := t#20ms); // BLINK
// fb_write_negative_el(
//     Execute := fb_blink_5.OUT,
//     ParameterNumber := FP_S_0_0050,
//     Value := r_limit_el_down,
//     Axis := drive3); // MB_WriteRealParameter

// NETWORK 11 (disabled)
//   axisdata[3].Axis_Inbb: A-0-0021.13 -RD- Axis is ready for power to the amplifier (bb)
//   FP_S_0_0049: Positive position limit value
//   drive3: Real axis "Drive3" with axis number 3
// fb_blink_6(ENABLE := NOT gc_b_sim_on AND axisdata[3].Axis_Inbb, TIMELOW := t#20ms, TIMEHIGH := t#20ms); // BLINK
// fb_write_positive_el(
//     Execute := fb_blink_6.OUT,
//     ParameterNumber := FP_S_0_0049,
//     Value := r_limit_el_up,
//     Axis := drive3); // MB_WriteRealParameter

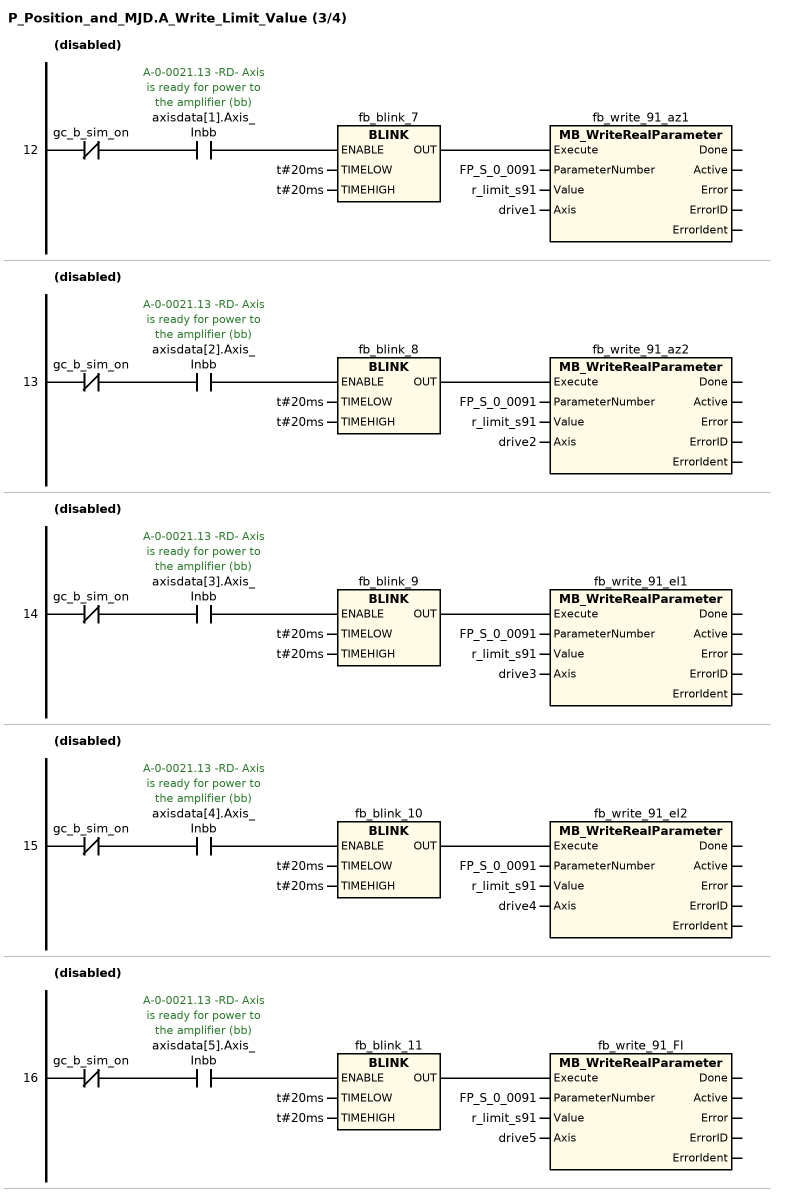
// NETWORK 12 (disabled)
//   axisdata[1].Axis_Inbb: A-0-0021.13 -RD- Axis is ready for power to the amplifier (bb)
//   FP_S_0_0091: Bipolar velocity limit value
//   drive1: Real axis "Drive1" with axis number 1
// fb_blink_7(ENABLE := NOT gc_b_sim_on AND axisdata[1].Axis_Inbb, TIMELOW := t#20ms, TIMEHIGH := t#20ms); // BLINK
// fb_write_91_az1(
//     Execute := fb_blink_7.OUT,
//     ParameterNumber := FP_S_0_0091,
//     Value := r_limit_s91,
//     Axis := drive1); // MB_WriteRealParameter

// NETWORK 13 (disabled)
//   axisdata[2].Axis_Inbb: A-0-0021.13 -RD- Axis is ready for power to the amplifier (bb)
//   FP_S_0_0091: Bipolar velocity limit value
//   drive2: Real axis "Drive2" with axis number 2
// fb_blink_8(ENABLE := NOT gc_b_sim_on AND axisdata[2].Axis_Inbb, TIMELOW := t#20ms, TIMEHIGH := t#20ms); // BLINK
// fb_write_91_az2(
//     Execute := fb_blink_8.OUT,
//     ParameterNumber := FP_S_0_0091,
//     Value := r_limit_s91,
//     Axis := drive2); // MB_WriteRealParameter

// NETWORK 14 (disabled)
//   axisdata[3].Axis_Inbb: A-0-0021.13 -RD- Axis is ready for power to the amplifier (bb)
//   FP_S_0_0091: Bipolar velocity limit value
//   drive3: Real axis "Drive3" with axis number 3
// fb_blink_9(ENABLE := NOT gc_b_sim_on AND axisdata[3].Axis_Inbb, TIMELOW := t#20ms, TIMEHIGH := t#20ms); // BLINK
// fb_write_91_el1(
//     Execute := fb_blink_9.OUT,
//     ParameterNumber := FP_S_0_0091,
//     Value := r_limit_s91,
//     Axis := drive3); // MB_WriteRealParameter

// NETWORK 15 (disabled)
//   axisdata[4].Axis_Inbb: A-0-0021.13 -RD- Axis is ready for power to the amplifier (bb)
//   FP_S_0_0091: Bipolar velocity limit value
//   drive4: Real axis "Drive4" with axis number 4
// fb_blink_10(ENABLE := NOT gc_b_sim_on AND axisdata[4].Axis_Inbb, TIMELOW := t#20ms, TIMEHIGH := t#20ms); // BLINK
// fb_write_91_el2(
//     Execute := fb_blink_10.OUT,
//     ParameterNumber := FP_S_0_0091,
//     Value := r_limit_s91,
//     Axis := drive4); // MB_WriteRealParameter

// NETWORK 16 (disabled)
//   axisdata[5].Axis_Inbb: A-0-0021.13 -RD- Axis is ready for power to the amplifier (bb)
//   FP_S_0_0091: Bipolar velocity limit value
//   drive5: Real axis "Drive5" with axis number 5
// fb_blink_11(ENABLE := NOT gc_b_sim_on AND axisdata[5].Axis_Inbb, TIMELOW := t#20ms, TIMEHIGH := t#20ms); // BLINK
// fb_write_91_FI(
//     Execute := fb_blink_11.OUT,
//     ParameterNumber := FP_S_0_0091,
//     Value := r_limit_s91,
//     Axis := drive5); // MB_WriteRealParameter

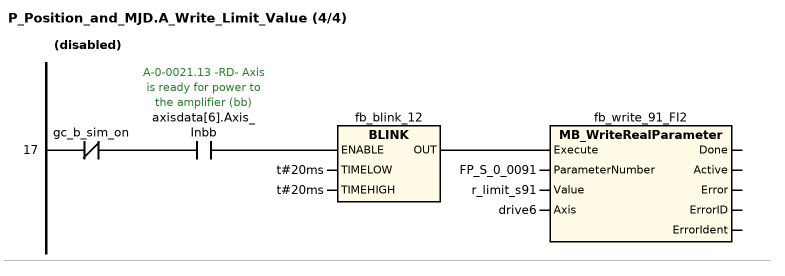
// NETWORK 17 (disabled)
//   axisdata[6].Axis_Inbb: A-0-0021.13 -RD- Axis is ready for power to the amplifier (bb)
//   FP_S_0_0091: Bipolar velocity limit value
//   drive6: Real axis "Drive6" with axis number 6
// fb_blink_12(ENABLE := NOT gc_b_sim_on AND axisdata[6].Axis_Inbb, TIMELOW := t#20ms, TIMEHIGH := t#20ms); // BLINK
// fb_write_91_FI2(
//     Execute := fb_blink_12.OUT,
//     ParameterNumber := FP_S_0_0091,
//     Value := r_limit_s91,
//     Axis := drive6); // MB_WriteRealParameter
END_ACTION

END_PROGRAM

// IndraMotionMlc1/Application/POUs/TCP/Message/deg2rad
FUNCTION deg2rad : LREAL
VAR_INPUT
degree_in:LREAL;	
END_VAR
VAR
END_VAR

deg2rad:=degree_in/180.0*3.1415926;

END_FUNCTION

// IndraMotionMlc1/Application/POUs/TCP/Message/Encoder_to_motor
FUNCTION Encoder_to_motor : LREAL
VAR_INPUT
	encoder_input:LREAL;
END_VAR
VAR
END_VAR

(*
Encoder_to_motor:=P1*EXPT(encoder_input+40,8)+P2*EXPT(encoder_input+40,7)+P3*EXPT(encoder_input+40,6)+P4*EXPT(encoder_input+40,5)
					+P5*EXPT(encoder_input+40,4)+P6*EXPT(encoder_input+40,3)+P7*EXPT(encoder_input+40,2)
						+P8*(encoder_input+40)+P9+1000000;
*)						
(*Encoder_to_motor:=P1*EXPT(encoder_input,9)+P2*EXPT(encoder_input,8)+P3*EXPT(encoder_input,7)+P4*EXPT(encoder_input,6)
					+P5*EXPT(encoder_input,5)+P6*EXPT(encoder_input,4)+P7*EXPT(encoder_input,3)+P8*EXPT(encoder_input,2)
						+P9*(encoder_input)+P10;
*)
					
Encoder_to_motor:=P1*EXPT(encoder_input,9)+P2*EXPT(encoder_input,8)+P3*EXPT(encoder_input,7)+P4*EXPT(encoder_input,6)
					+P5*EXPT(encoder_input,5)+P6*EXPT(encoder_input,4)+P7*EXPT(encoder_input,3)+P8*EXPT(encoder_input,2)
						+P9*(encoder_input)+P10-5441.92821;

END_FUNCTION

// IndraMotionMlc1/Application/POUs/Motion/POU_1MS
PROGRAM POU_1MS
VAR
	r_cycle_count: INT;
	R_TRIG_count: R_TRIG;
	R_TRIG_count_1: R_TRIG;
	r_cycle_count_1: INT;
	MB_AxisDistanceAccumulator_1: MB_AxisDistanceAccumulator;
	bDisenable: BOOL;
	
	btestStart: BOOL;
	rdistance: REAL;
	
	CTU_1: CTU;
	bReset: BOOL;
	bSTOPPPP: BOOL;
	iTestint: REAL;
	rdistancediff: REAL;
	rdiffdistance: REAL;
	rOldDistance: REAL;
	bHometest: BOOL;
	MB_WriteRealParameter_1: MB_WriteRealParameter;
	rIniEncoderPos: REAL;

	R_TRIG_IniPos: R_TRIG;
	bStartRecord: BOOL;
	R_TRIG_condition: R_TRIG;
	teetet: BOOL;
	TON_1: TON;
	rAxis3ActVel: REAL;
	rSetAxis3Vel: REAL;
	
	R_TRIG_VEL: R_TRIG;
	test_motor_degree: LREAL;
	test_encoder: LREAL;
	
	postion_vel_array:ARRAY[1..201] OF LREAL;
	MJD_vel_array:ARRAY[1..201] OF LREAL;
	pos_vel_avg_array:ARRAY[1..181] OF LREAL;
	position_vel_i:INT:=0;
	position_vel_avg_i:INT:=0;
	position_vel_i_before:INT;
	r_temp1_pos:LREAL;
	r_temp1_mjd:LREAL;
	i_temp:INT;
	sum_vel:LREAL;


	i_avg_1:INT:=0;
	i_avg_2:INT:=0;
	i_avg_3:INT:=0;
	temp_vel_avg_array:ARRAY[1..21] OF LREAL;
	sum_temp_vel:LREAL;
	test1_temp:LREAL;
	r_new_cmd_pos:LREAL;
	r_new_cmd_pos_motor:LREAL;
	r_new_cmd_pos_motor_relative:LREAL;
	R_TRIG_pos_done:R_TRIG;
	R_TRIG_pos_done_2:R_TRIG;
	R_TRIG_pos_done_3:R_TRIG;
	R_TRIG_pos_done_4:R_TRIG;
	R_TRIG_pos_done_5:R_TRIG;
	R_TRIG_pos_done_6:R_TRIG;
	R_TRIG_pos_done_7:R_TRIG;
	R_TRIG_pos_done_8:R_TRIG;
	R_TRIG_pos_done_9:R_TRIG;
	R_TRIG_pos_done_10:R_TRIG;
	ton_pos2:TON;
	
	i_closeloop_max:INT:=10;
	i_time:INT:=0;
	r_difference:LREAL;
	test_POWER_EL: BOOL;
	vel_blink:Util.BLINK;
	rSPEED1: LREAL;
	ton_start_adjust_vel:TON;
	r_trig_start_adjust_vel: R_TRIG;
	r_vel_el_1:LREAL;
	
	vel_freq:LREAL;
	T_period:LREAL:=1;
	temp_t:LREAL:=0.0;
	start_to_freq:BOOL;
	temp_i:INT:=0;
	
	b_test_freq_resp: BOOL;
	b_in_normal_mode: BOOL := TRUE;
	b_test_pos_freq: BOOL;
	
	Frequency_vel:LREAL:=0.4;
	b_test_random_array: BOOL;
	start_to_random_array: BOOL;
	i_random_count:DINT:=0;
	random_gain: LREAL:=1;
	i_test_count:DINT:=0;
	vel_random_array:LREAL;
	vel_random_array1:LREAL;
	test_1: BOOL;
	ML_WriteCyclicVelocity_0: MC_MoveVelocity;
	test_vel: LREAL;
	test_move_done: BOOL;
	R_TRIG_0: R_TRIG;
	r_motorencoder_11: LREAL;
	r_motorencoder_22: LREAL;
	FB_readmotorencoder11: MB_ReadRealParameter;
	FB_readmotorencoder22: MB_ReadRealParameter;
	R_TRIG_1: R_TRIG;
	temp_t1: LREAL:=0.0;
	BLINK_0: BLINK;
	b_test_freq_torque: BOOL;
	r_unbalance_torque:LREAL;
	
	r_freq_test_velmode_A:LREAL:=100;
	
	torque_freq:LREAL;
	
	b_test_az_freq_torque: BOOL;
	test_torque: LREAL;
	
	r_freq_test_torquemode_A:REAL:=60;
	b_test_az_frequence:BOOL;
	b_test_el_frequence:BOOL;
	FB_read1: MB_ReadRealParameter;
	r_drive3_s80: LREAL;
	FB_read2: MB_ReadRealParameter;
	r_drive3_s81: LREAL;
	FB_read3: MB_ReadRealParameter;
	r_drive3_p49: LREAL;
	test_2: BOOL;
	ML_OpenCyclicVelocityChannel_0: ML_OpenCyclicVelocityChannel;
	b_open_channel_el_vel_done: BOOL;
	
	FB_write_cycle_el_vel: ML_WriteCyclicVelocity;
	b_write_el_vel_done: BOOL;
	R_el_cycle_vel: r_trig;
	K_gear_ratio_vel:LREAL;
	
	AZ1_actualvelocity:LREAL;
	AZ2_actualvelocity:LREAL;
END_VAR


(*****************测试谐振**************)
(*****************第一步，打开trace程序，***
（******方位 Trace_AZ_freq_res,俯仰 Trace_EL_freq_res**************)
(*****************第二步，设定扫频幅值**************)
//r_freq_test_torquemode_A;
(***********第三步，选定要测试的轴，方位和俯仰不要同时选中**********)
//b_test_az_frequence;
//b_test_el_frequence;

(*****************第四步，在软件界面转动到测试位置，再用速度模式转动轴，***
（******方位速度为0.1度/s,俯仰为0.03度/s**************)
(*****************第五步，trace重新开始记录**************)
(*****************第六步，启动力矩扫频**************)
//b_test_freq_torque;
(**********第七步，结束扫频，trace停止记录，存盘，停止力矩扫频，轴停止速度*******)
//b_test_freq_torque;



AZ1_actualvelocity := axisdata[1].rActualVelocity_i * 3000;
AZ2_actualvelocity := axisdata[2].rActualVelocity_i * 3000;




IF b_test_az_frequence AND b_test_el_frequence THEN
	b_test_az_frequence:=FALSE;
	b_test_el_frequence:=FALSE;
END_IF


//axisdata[3].rActualPosition_i;

	position_vel_i:= position_vel_i+1;
	IF position_vel_i>200 THEN
		position_vel_i:=1;
	END_IF
	postion_vel_array[position_vel_i]:=r_pos_el;
	MJD_vel_array[position_vel_i]:=lr_MJD_current;
	
	position_vel_i_before:=position_vel_i-100;
	IF position_vel_i_before<0 THEN
		position_vel_i_before:=position_vel_i_before+200;
	END_IF
	IF position_vel_i_before=0 THEN
		position_vel_i_before:=200;
	END_IF
		
	r_temp1_pos:=postion_vel_array[position_vel_i]-postion_vel_array[position_vel_i_before];
	r_temp1_mjd:=(MJD_vel_array[position_vel_i]-MJD_vel_array[position_vel_i_before])*86400;
	IF r_temp1_mjd= 0 THEN
		r_temp1_mjd :=1;
	END_IF
	position_vel_avg_i:=position_vel_avg_i+1;
	pos_vel_avg_array[position_vel_avg_i]:=r_temp1_pos/r_temp1_mjd;
	
	IF position_vel_avg_i = 180 THEN
		position_vel_avg_i:=0;
	END_IF
	
		sum_vel:=0;
	FOR i_temp :=1 TO 180 BY 1 DO
		sum_vel:=sum_vel+pos_vel_avg_array[i_temp];
	END_FOR
		r_vel_EL_temp:=sum_vel/180;
		
	i_avg_1:=i_avg_1+1;
	
	IF i_avg_1 =200 THEN
		i_avg_1:=0;
		i_avg_2:=i_avg_2+1;
		temp_vel_avg_array[i_avg_2]:=r_vel_EL_temp;
		IF i_avg_2>20 THEN
			i_avg_2:=0;
		END_IF		
	END_IF
	
		sum_temp_vel:=0;
	FOR i_avg_3 :=1 TO 20 BY 1 DO
		sum_temp_vel:=sum_temp_vel+temp_vel_avg_array[i_avg_3];
	END_FOR
		r_vel_EL:=sum_temp_vel/20;
	

		
	
	
//	r_vel_EL:=r_temp1_pos/r_temp1_mjd;
//	r_vel_EL:=(postion_vel_array[position_vel_i]-postion_vel_array[position_vel_i_before])/(MJD_vel_array[position_vel_i]-MJD_vel_array[position_vel_i_before])/86400;
	
	
	
	test_motor_degree:=Encoder_to_motor(test_encoder);
 
	//俯仰电机实时位置	
	r_pos_motor3:=axisdata[3].rActualPosition_i;	
	
	//俯仰电机位置累计
    rPosdiff:=RIL_Utilities.IL_GetModuloType04((axisdata[3].rActualPosition_i-roldposition),210000);
	//rPosdiff:=r_pos_motor3-roldposition;
	roldposition:=r_pos_motor3;
	r_length:=r_length+rPosdiff;
	
	CTU_1(CU:=axisdata[3].rActualPosition_i>180 , RESET:= bReset, PV:=10000 , Q=> , CV=> );
	CTU_1.CV;
	//测量Delta杆长值
	r_length_count := r_length/360/16.8*25;	
	
	//理论杆长
	Inir_Length:=SQRT(2984.1*2984.1+3150.6*3150.6-2*2984.1*3150.6*COS(r_pos_el*3.1415926/180));
	
	MB_AxisDistanceAccumulator_1(
	Enable:= bDisenable, 
	TotalDistance:= 1000000, 
	InOperation=> , 
	Error=> , 
	ErrorID=> , 
	ErrorIdent=> , 
	DistanceReached=> , 
	AccumulatedDistance=> r_length_Distance, 
	Axis:= Drive3);
/////////////**********上电设置编码器位置************////////////	
	R_TRIG_condition(CLK:=NOT TechBase.ImcStatus.Diag.Error 
							AND NOT arAxisStatus_gb[3].Admin.MODE_AH 
								AND ML_Base.AxisData[3].Axis_Inbb
									AND NOT bStartRecord, Q=> );
	IF  R_TRIG_condition.Q OR teetet  THEN 
		bHometest:=FALSE;
	END_IF
		MB_WriteRealParameter_1(
		Execute:= bHometest, 
		Done=> , 
		Active=> , 
		Error=> , 
		ErrorID=> , 
		ErrorIdent=> , 
		ParameterNumber:= ML_Base.FP_S_0_0052, 
		Value:= r_pos_motor3_Ini, 
		Axis:=Drive3 );	
	arAxisCtrl_gb[3].Admin.SetAbsRef:=MB_WriteRealParameter_1.Done;
		TON_1(IN:= MB_WriteRealParameter_1.Done, PT:=T#3S , Q=> , ET=> );
	//	R_TRIG_IniPos(CLK:= TON_1.Q, Q=> );
		IF TON_1.Q THEN 
			bStartRecord:=TRUE;
			bHometest:=FALSE;
		END_IF
		IF bStartRecord THEN
			r_pos_motor3_Ini:=axisdata[3].rActualPosition_i;
		END_IF
/////////////////**************************//////////////////////////	
 (*SIN_Curve  	
   iTestint:=iTestint+0.05;
   rdistance:=3600*SIN(iTestint*3.1415926/180);
   rdiffdistance:=rdistance-rOldDistance;
   rOldDistance:=rdistance;
   *) 
   
R_TRIG_VEL(CLK:=P_TCP_with_SCC.b_scc_vel1 , Q=> );	
IF R_TRIG_VEL.Q THEN 
	b_scc_vel1_temp:=TRUE;
END_IF

R_TRIG_pos_done(CLK:=arAxisStatus_gb[Drive3.AxisNo].Admin.CmdDone , Q=> );	
IF R_TRIG_pos_done.Q THEN 
	b_first_pos_done:=TRUE;
END_IF

R_TRIG_pos_done_2(CLK:=(arAxisStatus_gb[Drive3.AxisNo].Admin.CmdDone AND i_adjust_count=1) , Q=> );	
IF R_TRIG_pos_done_2.Q THEN 
	b_second_pos_done:=TRUE;
END_IF

R_TRIG_pos_done_3(CLK:=(arAxisStatus_gb[Drive3.AxisNo].Admin.CmdDone AND i_adjust_count=2) , Q=> );	
IF R_TRIG_pos_done_3.Q THEN 
	b_3rd_pos_done:=TRUE;
END_IF

R_TRIG_pos_done_4(CLK:=(arAxisStatus_gb[Drive3.AxisNo].Admin.CmdDone AND i_adjust_count=3) , Q=> );	
IF R_TRIG_pos_done_4.Q THEN 
	b_4th_pos_done:=TRUE;
END_IF

R_TRIG_pos_done_5(CLK:=(arAxisStatus_gb[Drive3.AxisNo].Admin.CmdDone AND i_adjust_count=4) , Q=> );	
IF R_TRIG_pos_done_5.Q THEN 
	b_5th_pos_done:=TRUE;
END_IF

R_TRIG_pos_done_6(CLK:=(arAxisStatus_gb[Drive3.AxisNo].Admin.CmdDone AND i_adjust_count=5) , Q=> );	
IF R_TRIG_pos_done_6.Q THEN 
	b_6th_pos_done:=TRUE;
END_IF

R_TRIG_pos_done_7(CLK:=(arAxisStatus_gb[Drive3.AxisNo].Admin.CmdDone AND i_adjust_count=6) , Q=> );	
IF R_TRIG_pos_done_7.Q THEN 
	b_7th_pos_done:=TRUE;
END_IF

R_TRIG_pos_done_8(CLK:=(arAxisStatus_gb[Drive3.AxisNo].Admin.CmdDone AND i_adjust_count=7) , Q=> );	
IF R_TRIG_pos_done_8.Q THEN 
	b_8th_pos_done:=TRUE;
END_IF

R_TRIG_pos_done_9(CLK:=(arAxisStatus_gb[Drive3.AxisNo].Admin.CmdDone AND i_adjust_count=8) , Q=> );	
IF R_TRIG_pos_done_9.Q THEN 
	b_9th_pos_done:=TRUE;
END_IF

R_TRIG_pos_done_10(CLK:=(arAxisStatus_gb[Drive3.AxisNo].Admin.CmdDone AND i_adjust_count=9) , Q=> );	
IF R_TRIG_pos_done_10.Q THEN 
	b_10th_pos_done:=TRUE;
END_IF

ton_pos2(IN:=b_second_pos_done,PT:=T#2S);
IF ton_pos2.Q THEN
adjust_delay:=TRUE;
END_IF

i_time:=i_time+1;
IF i_time>500 THEN
	i_time:=0;
END_IF

//IF i_time = 50 THEN
	IF TRUE AND i_time = 50 THEN
	r_difference:=ABS(r_goto_el_I-r_pos_el);

IF b_in_positionMode  AND b_first_pos_done AND i_adjust_count=0 AND r_difference>0.0005 THEN

	r_new_cmd_pos:=2*r_goto_el_I-r_pos_el;
	r_new_cmd_pos_motor:=Encoder_to_motor(r_new_cmd_pos);
	r_new_cmd_pos_motor_relative:=Encoder_to_motor(r_goto_el_I)-Encoder_to_motor(ML_Base.AxisData[11].rActualPosition_i);
	r_goto_el_abs:=r_new_cmd_pos_motor;
	r_goto_el:=r_new_cmd_pos_motor_relative;
	b_in_positionMode:=FALSE;
	b_first_pos_done:=FALSE;
	b_second_pos_done:=FALSE;
	b_3rd_pos_done:=FALSE;
	b_4th_pos_done:=FALSE;
	b_5th_pos_done:=FALSE;
	b_6th_pos_done:=FALSE;
	b_7th_pos_done:=FALSE;
	b_8th_pos_done:=FALSE;
	b_9th_pos_done:=FALSE;
	b_10th_pos_done:=FALSE;
	i_adjust_count:=1;	
END_IF

IF i_adjust_count=1  AND b_second_pos_done AND  r_difference>0.0005 THEN

	r_new_cmd_pos:=2*r_goto_el_I-r_pos_el;
	r_new_cmd_pos_motor:=Encoder_to_motor(r_new_cmd_pos);
	r_new_cmd_pos_motor_relative:=Encoder_to_motor(r_goto_el_I)-Encoder_to_motor(ML_Base.AxisData[11].rActualPosition_i);
	r_goto_el_abs:=r_new_cmd_pos_motor;
	r_goto_el:=r_new_cmd_pos_motor_relative;
	b_in_positionMode:=FALSE;
	b_first_pos_done:=FALSE;
	b_second_pos_done:=FALSE;
	b_3rd_pos_done:=FALSE;
	b_4th_pos_done:=FALSE;
	b_5th_pos_done:=FALSE;
	b_6th_pos_done:=FALSE;
	b_7th_pos_done:=FALSE;
	b_8th_pos_done:=FALSE;
	b_9th_pos_done:=FALSE;
	b_10th_pos_done:=FALSE;
	adjust_delay:=FALSE;
	i_adjust_count:=2;
END_IF

IF i_adjust_count=2  AND b_3rd_pos_done AND r_difference>0.0005  THEN

	r_new_cmd_pos:=2*r_goto_el_I-r_pos_el;
	r_new_cmd_pos_motor:=Encoder_to_motor(r_new_cmd_pos);
	r_new_cmd_pos_motor_relative:=Encoder_to_motor(r_goto_el_I)-Encoder_to_motor(ML_Base.AxisData[11].rActualPosition_i);
	r_goto_el_abs:=r_new_cmd_pos_motor;
	r_goto_el:=r_new_cmd_pos_motor_relative;
	b_in_positionMode:=FALSE;
	b_first_pos_done:=FALSE;
	b_second_pos_done:=FALSE;
	b_3rd_pos_done:=FALSE;
	b_4th_pos_done:=FALSE;
	b_5th_pos_done:=FALSE;
	b_6th_pos_done:=FALSE;
	b_7th_pos_done:=FALSE;
	b_8th_pos_done:=FALSE;
	b_9th_pos_done:=FALSE;
	b_10th_pos_done:=FALSE;
	adjust_delay:=FALSE;
	i_adjust_count:=3;
END_IF

IF i_adjust_count=3  AND b_4th_pos_done AND r_difference>0.0005  THEN

	r_new_cmd_pos:=2*r_goto_el_I-r_pos_el;
	r_new_cmd_pos_motor:=Encoder_to_motor(r_new_cmd_pos);
	r_new_cmd_pos_motor_relative:=Encoder_to_motor(r_goto_el_I)-Encoder_to_motor(ML_Base.AxisData[11].rActualPosition_i);
	r_goto_el_abs:=r_new_cmd_pos_motor;
	r_goto_el:=r_new_cmd_pos_motor_relative;
	b_in_positionMode:=FALSE;
	b_first_pos_done:=FALSE;
	b_second_pos_done:=FALSE;
	b_3rd_pos_done:=FALSE;
	b_4th_pos_done:=FALSE;
	b_5th_pos_done:=FALSE;
	b_6th_pos_done:=FALSE;
	b_7th_pos_done:=FALSE;
	b_8th_pos_done:=FALSE;
	b_9th_pos_done:=FALSE;
	b_10th_pos_done:=FALSE;
	adjust_delay:=FALSE;
	i_adjust_count:=4;
END_IF

IF i_adjust_count=4  AND b_5th_pos_done AND r_difference>0.0005  THEN

	r_new_cmd_pos:=2*r_goto_el_I-r_pos_el;
	r_new_cmd_pos_motor:=Encoder_to_motor(r_new_cmd_pos);
	r_new_cmd_pos_motor_relative:=Encoder_to_motor(r_goto_el_I)-Encoder_to_motor(ML_Base.AxisData[11].rActualPosition_i);
	r_goto_el_abs:=r_new_cmd_pos_motor;
	r_goto_el:=r_new_cmd_pos_motor_relative;
	b_in_positionMode:=FALSE;
	b_first_pos_done:=FALSE;
	b_second_pos_done:=FALSE;
	b_3rd_pos_done:=FALSE;
	b_4th_pos_done:=FALSE;
	b_5th_pos_done:=FALSE;
	b_6th_pos_done:=FALSE;
	b_7th_pos_done:=FALSE;
	b_8th_pos_done:=FALSE;
	b_9th_pos_done:=FALSE;
	b_10th_pos_done:=FALSE;
	adjust_delay:=FALSE;
	i_adjust_count:=1;
END_IF
END_IF
(*
IF i_adjust_count=5  AND b_6th_pos_done THEN
	r_new_cmd_pos:=2*r_goto_el_I-r_pos_el;
	r_new_cmd_pos_motor:=Encoder_to_motor(r_new_cmd_pos);
	r_goto_el_abs:=r_new_cmd_pos_motor;
	b_in_positionMode:=FALSE;
	b_first_pos_done:=FALSE;
	b_second_pos_done:=FALSE;
	b_3rd_pos_done:=FALSE;
	b_4th_pos_done:=FALSE;
	b_5th_pos_done:=FALSE;
	b_6th_pos_done:=FALSE;
	b_7th_pos_done:=FALSE;
	b_8th_pos_done:=FALSE;
	b_9th_pos_done:=FALSE;
	b_10th_pos_done:=FALSE;
	adjust_delay:=FALSE;
	i_adjust_count:=6;
END_IF

IF i_adjust_count=6  AND b_7th_pos_done THEN
	r_new_cmd_pos:=2*r_goto_el_I-r_pos_el;
	r_new_cmd_pos_motor:=Encoder_to_motor(r_new_cmd_pos);
	r_goto_el_abs:=r_new_cmd_pos_motor;
	b_in_positionMode:=FALSE;
	b_first_pos_done:=FALSE;
	b_second_pos_done:=FALSE;
	b_3rd_pos_done:=FALSE;
	b_4th_pos_done:=FALSE;
	b_5th_pos_done:=FALSE;
	b_6th_pos_done:=FALSE;
	b_7th_pos_done:=FALSE;
	b_8th_pos_done:=FALSE;
	b_9th_pos_done:=FALSE;
	b_10th_pos_done:=FALSE;
	adjust_delay:=FALSE;
	i_adjust_count:=7;
END_IF

IF i_adjust_count=7  AND b_8th_pos_done THEN
	r_new_cmd_pos:=2*r_goto_el_I-r_pos_el;
	r_new_cmd_pos_motor:=Encoder_to_motor(r_new_cmd_pos);
	r_goto_el_abs:=r_new_cmd_pos_motor;
	b_in_positionMode:=FALSE;
	b_first_pos_done:=FALSE;
	b_second_pos_done:=FALSE;
	b_3rd_pos_done:=FALSE;
	b_4th_pos_done:=FALSE;
	b_5th_pos_done:=FALSE;
	b_6th_pos_done:=FALSE;
	b_7th_pos_done:=FALSE;
	b_8th_pos_done:=FALSE;
	b_9th_pos_done:=FALSE;
	b_10th_pos_done:=FALSE;
	adjust_delay:=FALSE;
	i_adjust_count:=8;
END_IF

IF i_adjust_count=8  AND b_9th_pos_done THEN
	r_new_cmd_pos:=2*r_goto_el_I-r_pos_el;
	r_new_cmd_pos_motor:=Encoder_to_motor(r_new_cmd_pos);
	r_goto_el_abs:=r_new_cmd_pos_motor;
	b_in_positionMode:=FALSE;
	b_first_pos_done:=FALSE;
	b_second_pos_done:=FALSE;
	b_3rd_pos_done:=FALSE;
	b_4th_pos_done:=FALSE;
	b_5th_pos_done:=FALSE;
	b_6th_pos_done:=FALSE;
	b_7th_pos_done:=FALSE;
	b_8th_pos_done:=FALSE;
	b_9th_pos_done:=FALSE;
	b_10th_pos_done:=FALSE;
	adjust_delay:=FALSE;
	i_adjust_count:=9;
END_IF

IF i_adjust_count=9  AND b_10th_pos_done THEN
	r_new_cmd_pos:=2*r_goto_el_I-r_pos_el;
	r_new_cmd_pos_motor:=Encoder_to_motor(r_new_cmd_pos);
	r_goto_el_abs:=r_new_cmd_pos_motor;
	b_in_positionMode:=FALSE;
	b_first_pos_done:=FALSE;
	b_second_pos_done:=FALSE;
	b_3rd_pos_done:=FALSE;
	b_4th_pos_done:=FALSE;
	b_5th_pos_done:=FALSE;
	b_6th_pos_done:=FALSE;
	b_7th_pos_done:=FALSE;
	b_8th_pos_done:=FALSE;
	b_9th_pos_done:=FALSE;
	b_10th_pos_done:=FALSE;
	adjust_delay:=FALSE;
	i_adjust_count:=10;
END_IF
*)
(*	
IF  arAxisStatus_gb[Drive3.AxisNo].Admin.CmdDone AND i_closeloop_count<i_closeloop_max THEN
	r_new_cmd_pos:=2*r_goto_el_I-r_pos_el;
	r_new_cmd_pos_motor:=Encoder_to_motor(r_new_cmd_pos);
	r_goto_el_abs:=r_new_cmd_pos_motor;
	arAxisStatus_gb[Drive3.AxisNo].Admin.CmdDone:=FALSE;
	i_closeloop_count:= i_closeloop_count+1;
END_IF
	IF i_closeloop_count>i_closeloop_max THEN
		i_closeloop_count:=i_closeloop_max;
	END_IF
*)
r_trig_start_adjust_vel(CLK:= b_scc_vel); 
IF r_trig_start_adjust_vel.Q THEN
	b_start_adjust_vel_temp:=TRUE;
END_IF

ton_start_adjust_vel(IN:=b_start_adjust_vel_temp,PT:=T#10S);
IF ton_start_adjust_vel.Q THEN
	b_start_adjust_vel_temp:=FALSE;
	b_start_adjust_vel:=TRUE;
END_IF

//	r_vel_el_1:= 0.00008*ML_Base.AxisData[11].rActualPosition_i*ML_Base.AxisData[11].rActualPosition_i - 0.0141*ML_Base.AxisData[11].rActualPosition_i + 1.6168;
//r_vel_el_1 := 0.0000000002*r_pos_el_v*r_pos_el_v*r_pos_el_v*r_pos_el_v*r_pos_el_v - 0.00000003*r_pos_el_v*r_pos_el_v*r_pos_el_v*r_pos_el_v + 0.000002*r_pos_el_v*r_pos_el_v*r_pos_el_v + 0.0001*r_pos_el_v*r_pos_el_v - 0.0187*r_pos_el_v + 1.6902;
r_vel_el_1 := -(0.00000000007173*r_pos_el_v*r_pos_el_v*r_pos_el_v*r_pos_el_v + 0.00000003909*r_pos_el_v*r_pos_el_v*r_pos_el_v - 0.00001355*r_pos_el_v*r_pos_el_v + 0.001506*r_pos_el_v - 0.1344)/0.1;
K_gear_ratio_vel:=K_gear_ratio/2000;
(**********************以下为伪随机序列测试模块***********************)
 IF start_to_random_array THEN
	 i_test_count:=i_test_count+1;
	 IF i_test_count=25 THEN
		 i_test_count:=0;
	 END_IF
	 
	 IF i_test_count=1 THEN
		 test_1:=FALSE;
		 test_move_done:=FALSE;
	 END_IF
	 
	 IF i_test_count =3 THEN
	 	i_random_count:=i_random_count+1;
		 vel_random_array:=track_table[i_random_count].Azimuth*random_gain;
		test_1:=TRUE;		 
	 END_IF
	 
	
	 IF i_random_count= i_End THEN 
		i_random_count:=0; 
	 END_IF	
 ELSE
		vel_random_array:=0;
		i_random_count:=0;
 END_IF	
 
(******************伪随机序列测试模块结束*********************) 


(*******************以下为谐振测试模块************************)
 IF start_to_freq OR b_test_freq_torque THEN
		T_period:=1/Frequency_vel;	 
 		IF temp_t<(20*T_period) THEN
			temp_t:=temp_t+0.001;
//			vel_freq:=r_freq_test_velmode_A*SIN(2*3.1415926*Frequency_vel*temp_t);
			torque_freq:=r_freq_test_torquemode_A*SIN(2*3.1415926*Frequency_vel*temp_t);
		ELSE
			temp_t:=0;
			temp_i:=temp_i+1;
			IF b_test_az_frequence THEN	
				IF Frequency_vel<1.5 THEN
					//Frequency_vel:=0.4+0.1*temp_i;
					Frequency_vel:=1+0.1*temp_i;
				ELSE
					//Frequency_vel:=1.5+0.05*(temp_i-11);
					Frequency_vel:=1.5+0.05*(temp_i-5);
				END_IF
			END_IF	
		
			IF b_test_el_frequence THEN	
				IF Frequency_vel<2 THEN
					Frequency_vel:=1+0.1*temp_i;
				ELSE
					Frequency_vel:=2+0.05*(temp_i-10);
				END_IF
			END_IF				
			IF Frequency_vel>3.0 THEN
				Frequency_vel:=3.0;
			END_IF
		END_IF
 ELSE
		temp_t:=0;
		temp_i:=0;
		IF b_test_az_frequence THEN
			//Frequency_vel:=0.4;
			Frequency_vel:=1.0;
		END_IF
		IF b_test_EL_frequence THEN
			Frequency_vel:=1.0;
		END_IF
		vel_freq:=0;
		torque_freq:=0;
 END_IF
(*************************谐振测试模块结束***********************)


 IF b_test_az_frequence AND b_test_freq_torque THEN
	ML_Base.AxisData[1].dwUserCmdDataB_q.REAL_:=torque_freq;
 END_IF
 
 
 
IF b_scc_vel1_temp OR b_test_freq_resp OR b_test_random_array OR b_test_freq_torque THEN
	
	IF b_in_normal_mode THEN 
		arAxisCtrl_gb[Drive3.AxisNo].VelMode.Velocity := P_TCP_with_SCC.r_vel_el/TO_REAL(r_vel_el_1);
	//	arAxisCtrl_gb[Drive3.AxisNo].VelMode.Velocity := P_TCP_with_SCC.r_vel_el*K_gear_ratio_vel;
		IF r_command_vel=0 THEN
		add_vel:=0;		
		END_IF	
	ELSE
		arAxisCtrl_gb[Drive3.AxisNo].VelMode.Velocity := TO_REAL(vel_freq);

		IF start_to_freq = FALSE AND start_to_random_array =FALSE THEN
			arAxisCtrl_gb[Drive3.AxisNo].VelMode.Velocity:=0;
		END_IF		
	END_IF
	
	IF b_test_freq_torque AND b_test_el_frequence THEN
		ML_Base.AxisData[3].dwUserCmdDataB_q.REAL_:=TO_REAL(torque_freq);
	END_IF
			
	arAxisCtrl_gb[Drive3.AxisNo].VelMode.Acceleration := 200;
	arAxisCtrl_gb[Drive3.AxisNo].VelMode.Deceleration := 100;
	arAxisCtrl_gb[Drive3.AxisNo].Admin._OpMode.en := ModeVel;
	
  
ELSIF b_scc_goto THEN
	r_following_1:=r_following_11;
	arAxisCtrl_gb[Drive3.AxisNo].Admin._OpMode.en := ModeCyclicVelocity; 
	b_write_el_vel:=TRUE;
(*

//	arAxisCtrl_gb[Drive3.AxisNo].PosMode.Position:=r_goto_el_abs;
	arAxisCtrl_gb[Drive3.AxisNo].PosMode.Distance := r_goto_el;
	arAxisCtrl_gb[Drive3.AxisNo].PosMode.Velocity := rSPEED;
	arAxisCtrl_gb[Drive3.AxisNo].PosMode.Acceleration := rACC;
	arAxisCtrl_gb[Drive3.AxisNo].PosMode.Deceleration := rDCC;
//	arAxisCtrl_gb[Drive3.AxisNo].Admin._OpMode.en := ModePosAbs;
	arAxisCtrl_gb[Drive3.AxisNo].Admin._OpMode.en := TechInterface.ModePosRel;
//	axisdata[Drive3.AxisNo].Axis_InPosition;
	arAxisStatus_gb[Drive3.AxisNo].Admin.CmdDone;
*)

			
ELSE
	arAxisCtrl_gb[Drive3.AxisNo].Admin._OpMode.en := ModeAB;
END_IF 


IF bSTOPPPP THEN
	arAxisCtrl_gb[Drive3.AxisNo].Admin._OpMode.en := ModeAB;
END_IF



////////////******天线恒定速度运行********///////////////////////\

	
rAxis3ActVel:=ML_Base.AxisData[11].rActualVelocity_i*60000;
ML_Base.AxisData[11].rActualPosition_i;
ML_Base.AxisData[11].rActualVelocity_i;


(*
R_TRIG_VEL(CLK:=P_TCP_with_SCC.b_scc_vel1 , Q=> );	
IF R_TRIG_VEL.Q THEN 
	b_scc_vel1_temp:=TRUE;
END_IF
IF b_scc_vel1_temp THEN
	arAxisCtrl_gb[Drive3.AxisNo].VelMode.Velocity := P_TCP_with_SCC.r_vel_el;
	arAxisCtrl_gb[Drive3.AxisNo].VelMode.Acceleration := 100;
	arAxisCtrl_gb[Drive3.AxisNo].VelMode.Deceleration := 100;
	arAxisCtrl_gb[Drive3.AxisNo].Admin._OpMode.en := ModeVel;
ELSE
		arAxisCtrl_gb[Drive3.AxisNo].Admin._OpMode.en := Modeab;
END_IF 
*)


POU_1MS.P_Move();

ACTION P_Move:
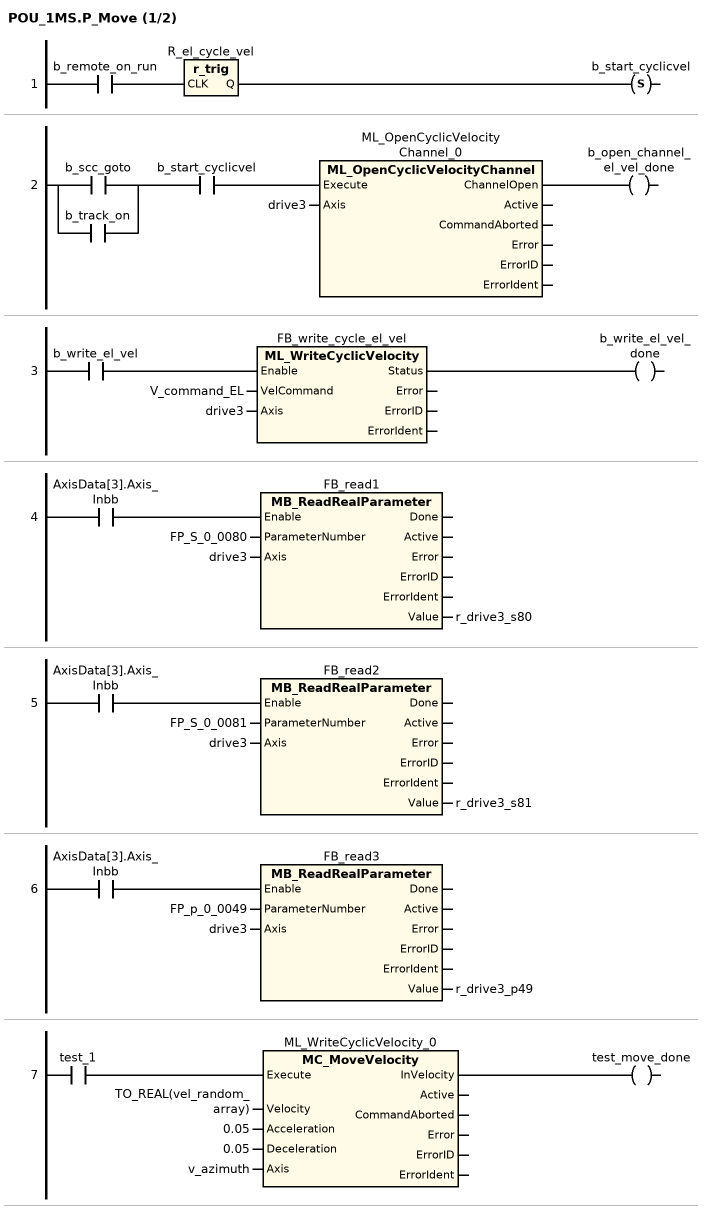
// NETWORK 1
R_el_cycle_vel(CLK := b_remote_on_run); // r_trig
b_start_cyclicvel S= R_el_cycle_vel.Q;

// NETWORK 2
ML_OpenCyclicVelocityChannel_0(Execute := (b_scc_goto OR b_track_on) AND b_start_cyclicvel, Axis := drive3); // ML_OpenCyclicVelocityChannel
b_open_channel_el_vel_done := ML_OpenCyclicVelocityChannel_0.ChannelOpen;

// NETWORK 3
FB_write_cycle_el_vel(Enable := b_write_el_vel, VelCommand := V_command_EL, Axis := drive3); // ML_WriteCyclicVelocity
b_write_el_vel_done := FB_write_cycle_el_vel.Status;

// NETWORK 4
//   FP_S_0_0080: Position feedback value 1
//   drive3: Real axis "Drive1" with axis number 1
FB_read1(
    Enable := AxisData[3].Axis_Inbb,
    ParameterNumber := FP_S_0_0080,
    Axis := drive3,
    Value => r_drive3_s80); // MB_ReadRealParameter

// NETWORK 5
//   FP_S_0_0081: Position feedback value 1
//   drive3: Real axis "Drive1" with axis number 1
FB_read2(
    Enable := AxisData[3].Axis_Inbb,
    ParameterNumber := FP_S_0_0081,
    Axis := drive3,
    Value => r_drive3_s81); // MB_ReadRealParameter

// NETWORK 6
//   FP_p_0_0049: Position feedback value 1
//   drive3: Real axis "Drive1" with axis number 1
FB_read3(
    Enable := AxisData[3].Axis_Inbb,
    ParameterNumber := FP_p_0_0049,
    Axis := drive3,
    Value => r_drive3_p49); // MB_ReadRealParameter

// NETWORK 7
ML_WriteCyclicVelocity_0(
    Execute := test_1,
    Velocity := TO_REAL(vel_random_array),
    Acceleration := 0.05,
    Deceleration := 0.05,
    Axis := v_azimuth); // MC_MoveVelocity
test_move_done := ML_WriteCyclicVelocity_0.InVelocity;

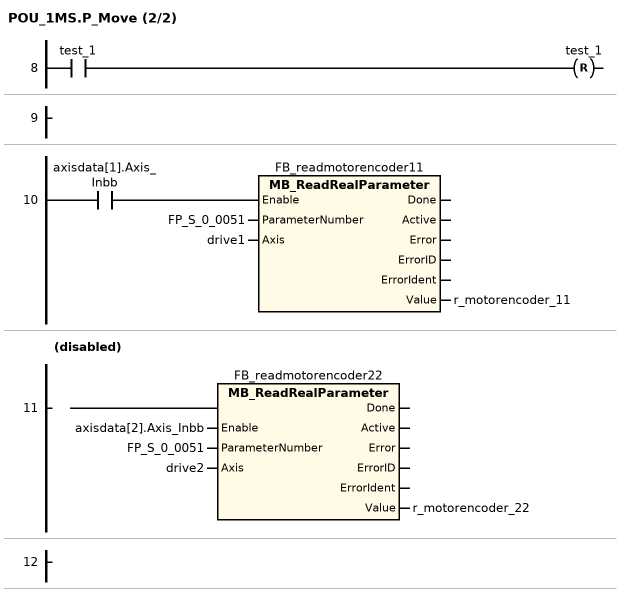
// NETWORK 8
test_1 R= test_1;

// NETWORK 9

// NETWORK 10
//   FP_S_0_0051: Position feedback value 1
//   drive1: Real axis "Drive1" with axis number 1
FB_readmotorencoder11(
    Enable := axisdata[1].Axis_Inbb,
    ParameterNumber := FP_S_0_0051,
    Axis := drive1,
    Value => r_motorencoder_11); // MB_ReadRealParameter

// NETWORK 11 (disabled)
//   axisdata[2].Axis_Inbb: A-0-0021.13 -RD- Axis is ready for power to the amplifier (bb)
//   FP_S_0_0051: Position feedback value 1
//   drive2: Real axis "Drive2" with axis number 2
// FB_readmotorencoder22(
//     Enable := axisdata[2].Axis_Inbb,
//     ParameterNumber := FP_S_0_0051,
//     Axis := drive2,
//     Value => r_motorencoder_22); // MB_ReadRealParameter

// NETWORK 12
END_ACTION

END_PROGRAM

// IndraMotionMlc1/Application/POUs/TCP/P_TCP_with_SCC
(*This program is built for TCP communication, receive the message from CSIRO,deal with the commands,and send the reply to CSIRO*)
PROGRAM P_TCP_with_SCC
VAR
(*<<<<<<<<<<<<<<<<<<<<<<<<<<<<<<<<<<<<<<<<<<<>>>>>>>>>>>>>>>>>>>>>>>>>>>>>>>>>>>>>*)
	b_receiving :BOOL;
	b_commanding: BOOL;
	b_sending: BOOL;
	str_MSG_Received:STRING(255);(*the received message*)
	fb_MSG_receive :FB_MSG;(*transfer the defined function block,FB_MSG*)
	fb_Trkval:FB_add_vector;(*transfer the defined function block,FB_add_vector*)
	b_Scc_PWR_on: BOOL;
	b_Scc_PWR_off: BOOL;
(*<<<<<<<<<<<<<<<<<<<<<<<<<<<<<<<<<<<<<<<<<<<CONNECTION>>>>>>>>>>>>>>>>>>>>>>>>>>>>>>>>>>>>>*)
	TCPConnection: IL_UDPSocketAsync;
	b_Server_Enable: BOOL:=TRUE;(*the enable of IL_TCPConnectionAsync*)
	di_Socket: DINT;(*the socket number*)
//	strIP: STRING;
	strIP: STRING:='10.160.63.111';
	b_Connection_done: BOOL;
(*<<<<<<<<<<<<<<<<<<<<<<<<<<<<<<<<<<<<<<<<<<<RECEIVE>>>>>>>>>>>>>>>>>>>>>>>>>>>>>>>>>>>>>*)
	TCPRecv:IL_UDPRecvfromAsync ;
	b_Recv_enable: BOOL;
	b_Recv_done: BOOL;
	str_Recv: STRING(255);
	di_ReceivedBytes: DINT;
(*<<<<<<<<<<<<<<<<<<<<<<<<<<<<<<<<<<<<<<<<<<<<SEND>>>>>>>>>>>>>>>>>>>>>>>>>>>>>>>>>>>>>*)
	TCPSend: IL_UDPSendtoAsync;
	b_Send_enable: BOOL;
	b_Send_done: BOOL;
	str_Send: STRING(1000);
	di_SentBytes: DINT;
(*<<<<<<<<<<<<<<<<<<<<<<<<<<<<<<<<<<<<<<<<<<<<<<<<<<<power>>>>>>>>>>>>>>>>>>>>>>>>>>>>>>>>>>>>*)
	ton_pow_off_az: TON;
	ton_pow_off_el: TON;
	ton_pow_off_FI: TON;
	rtrig_power_az: R_TRIG;
	rtrig_power_el: R_TRIG;
	rtrig_power_FI: R_TRIG;
	fb_ton_el: TON;
	fb_ton_FI: TON;
	rtrig_off_az: R_TRIG;
	rtrig_off_el: R_TRIG;
	rtrig_off_FI: R_TRIG;
	b_clear_err: BOOL;
	FB_clear_error_off: MB_WriteParameter;
	b_clear_off_done: BOOL;
	rtrig_err: R_TRIG;
	rtrig_clear_done: R_TRIG;
(*<<<<<<<<<<<<<<<<<<<<<<<<<<<<<<<<<<<<stop>>>>>>>>>>>>>>>>>>>>>>>>>>>>>*)
	b_stop1_done: BOOL;
	b_stop3_done: BOOL;
	b_stop5_done: BOOL;
	fb_scc_stop1: MC_Stop;
	fb_scc_stop3: MC_Stop;
	fb_scc_stop5: MC_Stop;
	rtrig_stop_az: R_TRIG;
	rtrig_stop_el: R_TRIG;
	rtrig_stop_FI: R_TRIG;
	b_stop_act_az: BOOL;
	b_stop_act_el: BOOL;
	b_stop_act_FI: BOOL;
	rtrig_reset_stop: R_TRIG;
(*<<<<<<<<<<<<<<<<<<<<<<<<<<<<<<<<<<<<<<<<<<<GOTO>>>>>>>>>>>>>>>>>>>>>>>>>>>>>>>>>>>>>>>>>>>*)


	fb_goto_Az: MC_MoveRelative;
	fb_goto_El: MC_MoveAbsolute;
	fb_goto_FI: MC_MoveRelative;
	b_active_AZ: BOOL;
	b_active_el: BOOL;
	b_active_FI: BOOL;
	rtrig_goto: R_TRIG;
(*K3STAT*)
	status_K3:DWORD;
(*add the function of close TCP function*)
	fb_tcp_close: IL_UDPCloseAsync;
	B_TCP_close: BOOL;
	b_TCP_close_done: BOOL;
	b_Recv_active: BOOL;
	i_counter_tcp:INT;
	rtrig_stop_stow: R_TRIG;
	Ftrig_goto: R_TRIG;
(*************vel**************)
r_vel_az:REAL;
r_vel_el:REAL;	
r_vel_FI:REAL;	

	
	rttig_vel: R_TRIG;
	b_scc_vel1: BOOL;
	fb_vel_az: MC_MoveVelocity;
	b_vel_az_done: BOOL;
	b_active_vel_az: BOOL;
	fb_vel_el: MC_MoveVelocity;
	b_active_vel_el: BOOL;
	b_vel_el_done: BOOL;
	fb_vel_FI: MC_MoveVelocity;
	b_active_vel_FI: BOOL;
	b_vel_FI_done: BOOL;
	fb_r_vel1: R_TRIG;
	fb_r_vel2: R_TRIG;
	fb_f_vel3: F_TRIG;
	fb_f_vel4: F_TRIG;
	fb_r_vel5: R_TRIG;
	fb_ton_vel: ton;
	str_concat: ARRAY[1..40] OF STRING(1000);(*数组及其类型的定义*)	
	Counter: INT;
	bWaiting4Connection: BOOL;
	bConnError: BOOL;
	diConnError: ERROR_CODE;
	ConnectError: ERROR_STRUCT;
i_counter_1s: INT:=0;	
	r_offset_az_I: REAL;
	r_offset_el_I: REAL;
	rtrig_power_power: R_TRIG;
	i_count:INT;
	
(*the status word for GSTAT*)	
	status_1:DWORD;
	status_2:DWORD;
	status_3:DWORD;
	status_4:DWORD;
	status_5:DWORD;
	status_6:DWORD;
(*the status code*)	
    drive_code1:STRING;
	drive_code2:STRING;
	drive_code3:STRING;
	drive_code4:STRING;
	drive_code5:STRING;
	drive_code6:STRING;

	
	vel_move_az: REAL:=0.3;
	vel_move_el: REAL:=0.167;
	vel_move_FI: REAL:=0.333;
	
	r_a0:REAL;
	v_a0:REAL;
	a_a0:REAL;
	t_difference:REAL;
	b_test:BOOL;
	
	r_az_pause_pos1:REAL;
	r_az_pause_pos2:REAL;
	r_az_pause_pos3:REAL;
	r_az_pause_pos4:REAL;
	r_az_pause_pos5:REAL;
	r_az_pause_pos6:REAL;
	r_az_pause_pos7:REAL;
	i_pause_temp:INT;
	
	fb_f_track_on:F_TRIG;
	b_not_track:BOOL;
	i_count_stop:INT;
	i_stop:INT;
	i_stop_1:INT;
	b_stop_TOA:BOOL;
	
	b_limit_az:BOOL;
	b_limit_el:BOOL;
	b_limit_FI:BOOL;
	
	fb_r_az_limit:r_trig;
	fb_r_el_limit:r_trig;
	fb_r_FI_limit:r_trig;
	
	i_new_cmd_dalay:DINT:=0;
	
	acc_mov_az: REAL;
	dcc_mov_az: REAL;
	vel_move_az_1: REAL;
	fb_start_goto_az: R_TRIG;
	b_moving: BOOL;
	fb_start_goto_az1: R_TRIG;
	fb_blink_move_az: BLINK;

	bTESTTTT: BOOL;
	fb_vel_el_1: MC_MoveVelocity;
	RTESTE: REAL;
	r_p1: LREAL;
	r_p0: LREAL;
	r_p2: LREAL;
	vel_stop_ton:TON;
	
	reply_count: DINT;
	TON_0: ton;
	FB_move_master_az1: MC_MoveAbsolute;
	b_Stop_Az: BOOL;
	b_start_goto_az_tcp: BOOL;
END_VAR


fb_f_track_on(clk:=b_track_on);

 IF b_goto_Az_done THEN
	b_step_running_az:=FALSE; 
 END_IF
 
 IF b_step_running_az=0 AND b_step_running_el=0 THEN
	 b_step_running:=0;
 END_IF
 IF b_step_running_az AND b_step_running_el THEN
	 b_step_running:=1;
 END_IF
 
 IF b_step_running OR b_offset_running THEN
	IF b_step_running THEN
	 r_step_count:=r_step_count_temp;
	END_IF 
	IF b_offset_running THEN
	 r_step_count:=r_offset_count_temp;
	END_IF 
 ELSE
	 r_step_count:=0;
 END_IF
	
 
 
 

	
IF fb_f_track_on.Q THEN
	b_not_track:=TRUE;	
END_IF

IF b_not_track AND i_num_stack_left=0 THEN
		i_start:=1;
		i_end:=1;
		track_table[1].TAIoffset:=0;
		FOR i_count:=1 TO i_total BY 1 DO
			track_table[i_count].TAIoffset:=0;
			track_table[i_count].Azimuth:= 0;
			track_table[i_count].Elevation:=0;
			//track_table[i_count].FeedIndexer:=0;
		END_FOR;
		(*track_table[1].MJD:=0;
		FOR i_count:=1 TO i_total BY 1 DO
			track_table[i_count].MJD:=0;
			track_table[i_count].Azimuth:= 0;
			track_table[i_count].Elevation:=0;
			track_table[i_count].FeedIndexer:=0;
		END_FOR;*)
END_IF

IF b_not_track AND  b_stop_TOA THEN
		i_start:=1;
		i_end:=1;
		track_table[1].TAIoffset:=0;
		FOR i_count:=1 TO i_total BY 1 DO
			track_table[i_count].TAIoffset:=0;
			track_table[i_count].Azimuth:= 0;
			track_table[i_count].Elevation:=0;
			//track_table[i_count].FeedIndexer:=0;
		END_FOR;
		(*track_table[1].MJD:=0;
		FOR i_count:=1 TO i_total BY 1 DO
			track_table[i_count].MJD:=0;
			track_table[i_count].Azimuth:= 0;
			track_table[i_count].Elevation:=0;
			track_table[i_count].FeedIndexer:=0;
		END_FOR; *)
		b_not_track:=FALSE;
		b_stop_TOA:=FALSE;
END_IF


IF i_start = i_end THEN
	b_on_track_mode:=FALSE;
	b_track_pause:=FALSE;
	b_permit_new_file:=TRUE;
END_IF



IF status_code1='A0160' OR status_code1='A0163' THEN
	drive_code1:='AF';
ELSIF  (status_code1='A0013' OR status_code1='A0012' ) AND axisdata[1].Axis_InAb THEN
	drive_code1:='Ab';
ELSIF  (status_code1='A0013' OR status_code1='A0012' ) AND axisdata[1].Axis_Inbb THEN 
	drive_code1:='bb';	
ELSE
	drive_code1:=status_code1;	
END_IF



IF status_code2='A0160' OR status_code2='A0163'THEN
	drive_code2:='AF';
ELSIF  (status_code2='A0013' OR status_code2='A0012' ) AND axisdata[2].Axis_InAb THEN
	drive_code2:='Ab';
ELSIF  (status_code2='A0013' OR status_code2='A0012' ) AND axisdata[2].Axis_Inbb THEN 
	drive_code2:='bb';	
ELSE
	drive_code2:=status_code2;	
END_IF

IF status_code1 = 'E2004' THEN
	drive_code1:=drive_code2;
END_IF

IF status_code3='A0160' OR status_code3='A0163' OR status_code3='A0161' OR status_code3='A0010' OR status_code3='A0101'THEN
	drive_code3:='AF';
ELSIF ( status_code3='A0013' OR status_code3='A0012' ) AND axisdata[3].Axis_InAb THEN
	drive_code3:='Ab';
ELSIF  (status_code3='A0013' OR status_code3='A0012' ) AND axisdata[3].Axis_Inbb THEN 
	drive_code3:='bb';	
ELSE
	drive_code3:=status_code3;	
END_IF

IF status_code4='A0160' OR status_code4='A0163'THEN
	drive_code4:='AF';
ELSIF  (status_code4='A0013' OR status_code4='A0012' ) AND axisdata[4].Axis_InAb THEN
	drive_code4:='Ab';
ELSIF  (status_code4='A0013' OR status_code4='A0012' ) AND axisdata[4].Axis_Inbb THEN 
	drive_code4:='bb';	
ELSE
	drive_code4:=status_code4;	
END_IF

IF status_code5='A0160' OR status_code5='A0163' THEN
	drive_code5:='AF';
ELSIF  (status_code5='A0013' OR status_code5='A0012' ) AND axisdata[5].Axis_InAb THEN
	drive_code5:='Ab';
ELSIF  (status_code5='A0013' OR status_code5='A0012' ) AND axisdata[5].Axis_Inbb THEN 
	drive_code5:='bb';	
ELSE
	drive_code5:=status_code5;	
END_IF

IF status_code6='A0160' OR status_code6='A0163' THEN
	drive_code6:='AF';
ELSIF  (status_code6='A0013' OR status_code6='A0012' )AND axisdata[6].Axis_InAb THEN
	drive_code6:='Ab';
ELSIF  (status_code6='A0013' OR status_code6='A0012' ) AND axisdata[6].Axis_Inbb THEN 
	drive_code6:='bb';	
ELSE
	drive_code6:=status_code6;	
END_IF

IF status_code1='E8029' OR status_code1='E8030' THEN
	b_limit_az:=TRUE;

ELSE
	b_limit_az:=FALSE;
END_IF

fb_r_az_limit(CLK:=b_limit_az);

IF fb_r_az_limit.Q THEN
	r_vel_az:=0;
	b_scc_vel:=TRUE;
END_IF

IF status_code3='E8029' OR status_code3='E8030' THEN
	b_limit_el:=TRUE;
ELSE
	b_limit_el:=FALSE;
END_IF

fb_r_el_limit(CLK:=b_limit_el);

IF fb_r_el_limit.Q THEN
	r_vel_el:=0;
	b_scc_vel:=TRUE;
END_IF

IF status_code5='E8029' OR status_code5='E8030' THEN
	b_limit_FI:=TRUE;
ELSE
	b_limit_FI:=FALSE;
END_IF

fb_r_FI_limit(CLK:=b_limit_FI);

IF fb_r_FI_limit.Q THEN
	r_vel_FI:=0;
	b_scc_vel:=TRUE;
END_IF



(*<<<<<<<<<<<<<<<<<<<<<<<<<<<<<master_status>>>>>>>>>>>>>>>>>>>>>>>>>>>>>>>>>>>>>>>>>>>>>>>>>>>>>>>*)
master_status.0:=(axisdata[1].Axis_InAb AND axisdata[2].Axis_InAb AND axisdata[3].Axis_InAb);
IF b_remote_on=TRUE THEN
	master_status.1:=0;
ELSE
	master_status.1:=1;
END_IF
IF b_DSdoor_ESTOP THEN
	master_status.2:=1;
ELSE
	master_status.2:=0;
END_IF

	master_status.3:=b_stow_lock;
	master_status.4:=(axisdata[1].Axis_Error OR axisdata[2].Axis_Error OR axisdata[3].Axis_Error);
	master_status.5:=b_stow_pin_limit_unlock;
	master_status.6:=b_stow_pin_limit_lock;
	
IF i_num_stack_left>9500 THEN
		master_status.7:=0;
	ELSE IF i_num_stack_left<1500 THEN
		master_status.7:=1;	
	END_IF
END_IF
	master_status.8:=0;
	master_status.9:=0;
	master_status.10:=0;



(*<<<<<<<<<<<<<<<<<<<<<<<<<<<<status_1>>>>>>>>>>>>>>>>>>>>>>>>>>>>>>>>>>>>>>>>>>>>>>>>>>>>>>>*)
status_1.0:=axisdata[1].Axis_InAb;
status_1.1:=axisdata[1].Axis_Power;
//status_1.1:=1;
status_1.2:=status_1.1;
status_1.3:=b_limit_ccw_az;
status_1.4:=b_limit_cw_az;
status_1.5:=axisdata[1].Axis_Error;
(*<<<<<<<<<<<<<<<<<<<<<<<<<<<<<status_2>>>>>>>>>>>>>>>>>>>>>>>>>>>>>>>>>>>>>>>>>>>>>>>>>>>>>>>*)
status_2.0:=axisdata[2].Axis_InAb;
status_2.1:=axisdata[2].Axis_Power;
//status_2.1:=1;
status_2.2:=status_2.1;
status_2.3:=b_limit_ccw_az;
status_2.4:=b_limit_cw_az;
status_2.5:=axisdata[2].Axis_Error;
(*<<<<<<<<<<<<<<<<<<<<<<<<<<<<<status_3>>>>>>>>>>>>>>>>>>>>>>>>>>>>>>>>>>>>>>>>>>>>>>>>>>>>>>>*)
status_3.0:=axisdata[3].Axis_InAb;
status_3.1:=axisdata[3].Axis_Power;
//status_3.1:=1;
status_3.2:=status_3.1;
status_3.3:=b_limit_ccw_el;
status_3.4:=b_limit_cw_el;
status_3.5:=axisdata[3].Axis_Error;

//axisdata[4].Axis_InAb:=axisdata[3].Axis_InAb;
//axisdata[5].Axis_InAb:=axisdata[3].Axis_InAb;
//axisdata[4].Axis_Power:=axisdata[3].Axis_Power;
//axisdata[5].Axis_Power:=axisdata[3].Axis_Power;

(*<<<<<<<<<<<<<<<<<<<<<<<<<<<<<status_4>>>>>>>>>>>>>>>>>>>>>>>>>>>>>>>>>>>>>>>>>>>>>>>>>>>>>>>*)
status_4.0:=axisdata[3].Axis_InAb;
status_4.1:=axisdata[3].Axis_Power;
//status_4.1:=1;
status_4.2:=status_4.1;
status_4.3:=b_limit_ccw_FI;
status_4.4:=b_limit_cw_FI;
status_4.5:=axisdata[3].Axis_Error;
(*<<<<<<<<<<<<<<<<<<<<<<<<<<<<<status_5>>>>>>>>>>>>>>>>>>>>>>>>>>>>>>>>>>>>>>>>>>>>>>>>>>>>>>>*)
status_5.0:=axisdata[3].Axis_InAb;
status_5.1:=axisdata[3].Axis_Power;
//status_5.1:=1;
status_5.2:=status_5.1;
status_5.3:=b_limit_ccw_FI;
status_5.4:=b_limit_cw_FI;
status_5.5:=axisdata[3].Axis_Error;





reply_count:=reply_count+1;
IF reply_count = 50 THEN	
	reply_count:=0;
END_IF

IF reply_count =10 OR reply_count =20 OR reply_count =30 OR reply_count =40 OR reply_count =50 THEN 

(*<<<<<<<<<<<<<<<<<<<<<<<<<<<<<concatenate STR_GSTAT>>>>>>>>>>>>>>>>>>>>>>>>>>>>>>>>>>>>>>>>>>>>>>>>>>>>>>>*)
				str_concat[1]:='OTHERSTATUS';
				str_concat[2]:=CONCAT(' ',LREAL_TO_STRING(lr_MJD_current));(*在track——running*)
				str_concat[3]:=CONCAT(' ',LREAL_TO_STRING(r_temp_motor1));(*在track——running*)
				str_concat[4]:=CONCAT(' ',LREAL_TO_STRING(r_temp_motor2));
    			str_concat[5]:=CONCAT(' ',LREAL_TO_STRING(r_temp_motor3));
 				str_concat[6]:=CONCAT(' ',LREAL_TO_STRING(r_temp_motor1));
				str_concat[7]:=CONCAT(' ',LREAL_TO_STRING(r_temp_motor2));	
				str_concat[8]:=CONCAT(' ',drive_code1);
				str_concat[9]:=CONCAT(' ',drive_code2);
				str_concat[10]:=CONCAT(' ',drive_code3);
				str_concat[11]:=CONCAT(' ',drive_code1);
				str_concat[12]:=CONCAT(' ',drive_code2);
				str_Send:='';(*for语句格式*)
				FOR Counter:=1 TO 12 BY 1 DO
					str_Send:=CONCAT(str_Send,str_concat[Counter]);
				END_FOR;

	ELSE				
(*<<<<<<<<<<<<<<<<<<<<<<<<<<<<<concatenate STR_GSTAT>>>>>>>>>>>>>>>>>>>>>>>>>>>>>>>>>>>>>>>>>>>>>>>>>>>>>>>*)
				str_concat[1]:='STATUS';
				str_concat[2]:=CONCAT(' ',LREAL_TO_STRING(lr_MJD_current));(*在track——running*)
				str_concat[3]:=CONCAT(' ',UINT_TO_STRING(i_Start));(*在track——running*)
				str_concat[4]:=CONCAT(' ',UINT_TO_STRING(i_End));(*在track——running*)
				str_concat[5]:=CONCAT(' ',INT_TO_STRING(i_num_stack_left));(*在track——running*)
				str_concat[6]:=CONCAT(' ',LREAL_TO_STRING(r_pos_az));
				str_concat[7]:=CONCAT(' ',LREAL_TO_STRING(r_pos_el));
 				str_concat[8]:=CONCAT(' ',LREAL_TO_STRING(r_pos_FI));
				str_concat[9]:=CONCAT(' ','1');   //MLC状态
    			str_concat[10]:=CONCAT(' ',DWORD_TO_STRING(master_status));
				str_concat[11]:=CONCAT(' ',LREAL_TO_STRING(r_following_1));
				str_concat[12]:=CONCAT(' ',LREAL_TO_STRING(r_following_3));
 				str_concat[13]:=CONCAT(' ',DINT_TO_STRING(r_step_count));
			  //str_concat[13]:=CONCAT(' ',REAL_TO_STRING(r_following_5));
				str_concat[14]:=CONCAT(' ',DWORD_TO_STRING(status_1));
				str_concat[15]:=CONCAT(' ',DWORD_TO_STRING(status_2));
				str_concat[16]:=CONCAT(' ',DWORD_TO_STRING(status_3));
				str_concat[17]:=CONCAT(' ',DWORD_TO_STRING(status_4));
				str_concat[18]:=CONCAT(' ',DWORD_TO_STRING(status_5));	
                str_concat[19]:=CONCAT(' ',LREAL_TO_STRING(r_current_1));
                str_concat[20]:=CONCAT(' ',LREAL_TO_STRING(i_speed_1));
                str_concat[21]:=CONCAT(' ',LREAL_TO_STRING(r_current_2));	
                str_concat[22]:=CONCAT(' ',LREAL_TO_STRING(i_speed_2));
                str_concat[23]:=CONCAT(' ',LREAL_TO_STRING(r_current_3));	
				str_concat[24]:=CONCAT(' ',LREAL_TO_STRING(i_speed_3));
				str_concat[25]:=CONCAT(' ',LREAL_TO_STRING(r_current_4));
				str_concat[26]:=CONCAT(' ',LREAL_TO_STRING(i_speed_4));
				str_concat[27]:=CONCAT(' ',LREAL_TO_STRING(r_current_5));
				str_concat[28]:=CONCAT(' ',LREAL_TO_STRING(i_speed_5));
				str_Send:='';(*for语句格式*)
				FOR Counter:=1 TO 28 BY 1 DO
					str_Send:=CONCAT(str_Send,str_concat[Counter]);
				END_FOR;
(*<<<<<<<<<<<<<<<<<<<<<<<<<<<if TCP is wrong,reset the TCP serve>>>>>>>>>>>>>>>>>>>>>>>>>>>>*)
END_IF				
				
				
(*<<<<<<<<<<<<<<<<<<<<<<<<<<<if TCP is wrong,reset the TCP serve>>>>>>>>>>>>>>>>>>>>>>>>>>>>*)
IF TCPConnection.Error=TRUE OR TCPRecv.Error=TRUE OR TCPSend.Error=TRUE THEN
	b_Server_Enable:=FALSE;
	b_Recv_enable:=FALSE;
	b_Send_enable:=FALSE;
ELSE
	b_Server_Enable:=TRUE;
END_IF

IF b_Connection_done = TRUE THEN
	i_counter_tcp := i_counter_tcp + 1;
END_IF;

(*
IF i_counter_tcp>2000 THEN
	B_TCP_close := TRUE;
	b_scc_enable_off := TRUE;
	b_scc_enable_on := FALSE;
	i_counter_tcp :=0;
ELSE
	B_TCP_close:= FALSE;
END_IF;
*)

P_TCP_with_SCC.Async_TCP();
P_TCP_with_SCC.A_RECV();
P_TCP_with_SCC.A_SEND();
(*<<<<<<<<<<<<<<<<<<<<<<<<<<<if TCP server is connected,a cycle is executed>>>>>>>>>>>>>>>>>>>>>>>>>>>>>>>>>>>>>>>>>>>>>*)
IF b_Connection_done=TRUE THEN
	IF  b_receiving=FALSE AND b_commanding=FALSE AND b_sending=FALSE AND b_Recv_enable=FALSE THEN
		b_Recv_enable:=TRUE;(*open recieve fuction*)
		P_TCP_with_SCC.A_RECV();
		b_receiving:=TRUE;
	END_IF;
(*<<<<<<<<<<<<<<<<<<<<<<<<<<<recieveing message>>>>>>>>>>>>>>>>>>>>>>>>>>>>>>>>>>>>>>>>>>>>>>>>>*)
	IF b_Recv_done=TRUE AND b_receiving=TRUE AND b_commanding=FALSE AND b_sending=FALSE THEN
		str_MSG_Received:=CONCAT(str_MSG_Received,LEFT(str_Recv,UDINT_TO_INT(di_ReceivedBytes)));
		fb_msg_receive(str_Message:=str_MSG_Received);
		str_MSG_Received:='';
		b_Recv_enable:=FALSE;
		P_TCP_with_SCC.A_RECV();
		b_receiving:=FALSE;
		b_commanding:=TRUE;
		i_counter_tcp :=0;
	END_IF
(*<<<<<<<<<<<<<<<<<<<<<<<<<<<<<<<<operating function>>>>>>>>>>>>>>>>>>>>>>>>>>>>>>>>>>>>>>>>>>>>>*)
	IF b_receiving=FALSE AND b_commanding=TRUE AND b_sending=FALSE THEN
(*<<<<<<<<<<<<<<<<<<<<<<<<<<<<<ENABLE>>>>>>>>>>>>>>>>>>>>>>>>>>>>>>>>>>>>>>>>>>>>>>>>>>>>>>>*)
		IF fb_msg_receive.Key='ENABLE'  THEN
			IF fb_msg_receive.P_value[1]='ON' THEN
				IF AXISDATA[1].Axis_InAb AND AXISDATA[3].Axis_InAb  THEN(*whether or not Power on*)
					b_off_write:=FALSE;
					b_on_write:=TRUE;
					b_SCC_enable_on:=TRUE;
					b_SCC_enable_off:=FALSE;
					IF b_remote_on THEN
					i_receive_cmd:=i_receive_cmd+1;
					i_excute_cmd:=i_excute_cmd+1;
					last_command:='05';
					END_IF
					str_Send:=F_RPL_1('',str_Send);
					b_commanding:=FALSE;
					b_sending:=TRUE;
				ELSE
					str_Send:=F_RPL_1('',str_Send);
					b_commanding:=FALSE;
					b_sending:=TRUE;
				END_IF;
			ELSIF fb_msg_receive.P_value[1]='OFF' THEN
					
					IF b_scc_vel1_temp THEN
					b_start_adjust_vel:=FALSE;
					b_start_adjust_vel_temp:=FALSE;
					r_vel_az:=0;
					r_vel_el:=0;
					b_scc_vel:=TRUE;
					P_TCP_with_SCC.A_SCC_GOTO();
					vel_stop_ton(IN := b_scc_vel, PT:= T#3S);
					vel_stop_ton.ET;
					IF vel_stop_ton.Q THEN
						b_scc_vel1_temp:=FALSE;
					b_on_write:=FALSE;
					b_off_write:=TRUE;
					b_scc_vel:=FALSE;
					b_scc_enable_off:=TRUE;
					b_SCC_enable_on:=FALSE;
					b_scc_goto:=FALSE;
					b_active_AZ:=FALSE;
					b_active_EL:=FALSE;
					b_active_FI:=FALSE;
					b_goto_Az_done:=FALSE;
					b_goto_EL_done:=FALSE;
					b_goto_FI_done:=FALSE;
					b_SCC_STOP:=FALSE;
					b_stop_act_az:=FALSE;
					b_stop_act_el:=FALSE;
					b_stop_act_FI:=FALSE;
					b_stop1_done:=FALSE;
					b_stop3_done:=FALSE;
					b_stop5_done:=FALSE;
					b_scc_maintain:=FALSE;
					b_scc_stow:=FALSE;
					b_write_az:=FALSE;
					b_write_el:=FALSE;
					b_write_FI:=FALSE;
					b_write_az_done:=FALSE;
					b_write_el_done:=FALSE;
					b_write_FI_done:=FALSE;
					b_open_channel_az:=FALSE;
					b_open_channel_el:=FALSE;
					b_open_channel_FI:=FALSE;
					b_open_channel_az_done:=FALSE;
					b_open_channel_el_done:=FALSE;
					b_open_channel_FI_done:=FALSE;
					b_move_0_done:=FALSE;
					b_move_20_done:=FALSE;
					b_lock_off:=FALSE;
					b_Track_Pause:=FALSE;
					b_track_on:=FALSE;
					b_on_track_mode:=FALSE;
					b_track_on_first:=FALSE;
					B_encoder_home_d1:=FALSE;
					B_encoder_home_d5:=FALSE;
					b_home_d1:=FALSE;
					b_home_d5:=FALSE;
					b_stop_TOA:=FALSE;
					b_move_to_start1:=FALSE;
					b_move_to_start5:=FALSE;
					b_in_positionMode:=FALSE;
					i_adjust_count:=0;
					b_first_pos_done:=FALSE;
					b_second_pos_done:=FALSE;
					b_3rd_pos_done:=FALSE;
					b_4th_pos_done:=FALSE;
					b_5th_pos_done:=FALSE;
					b_6th_pos_done:=FALSE;
					b_7th_pos_done:=FALSE;
					b_8th_pos_done:=FALSE;
					b_9th_pos_done:=FALSE;
					b_10th_pos_done:=FALSE;
					adjust_delay:=FALSE;
					i_closeloop_count:=0;
					END_IF		
					END_IF
					b_start_adjust_vel:=FALSE;
					b_start_adjust_vel_temp:=FALSE;
					b_scc_vel1_temp:=FALSE;
					b_on_write:=FALSE;
					b_off_write:=TRUE;
					b_scc_vel:=FALSE;
					b_scc_enable_off:=TRUE;
					b_SCC_enable_on:=FALSE;
					b_scc_goto:=FALSE;
					b_active_AZ:=FALSE;
					b_active_EL:=FALSE;
					b_active_FI:=FALSE;
					b_goto_Az_done:=FALSE;
					b_goto_EL_done:=FALSE;
					b_goto_FI_done:=FALSE;
					b_SCC_STOP:=FALSE;
					b_stop_act_az:=FALSE;
					b_stop_act_el:=FALSE;
					b_stop_act_FI:=FALSE;
					b_stop1_done:=FALSE;
					b_stop3_done:=FALSE;
					b_stop5_done:=FALSE;
					b_scc_maintain:=FALSE;
					b_scc_stow:=FALSE;
					b_write_az:=FALSE;
					b_write_el:=FALSE;
					b_write_FI:=FALSE;
					b_write_az_done:=FALSE;
					b_write_el_done:=FALSE;
					b_write_FI_done:=FALSE;
					b_open_channel_az:=FALSE;
					b_open_channel_el:=FALSE;
					b_open_channel_FI:=FALSE;
					b_open_channel_az_done:=FALSE;
					b_open_channel_el_done:=FALSE;
					b_open_channel_FI_done:=FALSE;
					b_move_0_done:=FALSE;
					b_move_20_done:=FALSE;
					b_lock_off:=FALSE;
					b_Track_Pause:=FALSE;
					b_track_on:=FALSE;
					b_on_track_mode:=FALSE;
					b_track_on_first:=FALSE;
					B_encoder_home_d1:=FALSE;
					B_encoder_home_d5:=FALSE;
					b_home_d1:=FALSE;
					b_home_d5:=FALSE;
					b_stop_TOA:=FALSE;
					b_move_to_start1:=FALSE;
					b_move_to_start5:=FALSE;
					b_in_positionMode:=FALSE;
					i_adjust_count:=0;
					b_first_pos_done:=FALSE;
					b_second_pos_done:=FALSE;
					b_3rd_pos_done:=FALSE;
					b_4th_pos_done:=FALSE;
					b_5th_pos_done:=FALSE;
					b_6th_pos_done:=FALSE;
					b_7th_pos_done:=FALSE;
					b_8th_pos_done:=FALSE;
					b_9th_pos_done:=FALSE;
					b_10th_pos_done:=FALSE;
					b_SCC_STOP:=FALSE;
					adjust_delay:=FALSE;
					i_closeloop_count:=0;
					lockstand:=TRUE;
					V_LastSpeed:=0;
					V_LastOutput:=0;
					dIntegralSpeed:= 0;	
					V_command_EL:=0;
					b_start_cyclicvel:=FALSE;
					b_write_el_vel:=FALSE;	
					b_step_running:=0;
					b_step_running_az:=0;
					b_step_running_el:=0;
					r_step_count:=0;
					r_step_count_temp:=0;
					b_offset_running:=0;
					r_offset_count_temp:=0;
					r_offset_count:=0;	
					r_offset_az:=0;
					r_offset_el:=0;
					V_LastOutput:=0;
					V_command_EL:=0;
					Pos_EL_error:=0;
					r_test_offset_el:=0;
					r_test_offset_az:=0;
					dIntegralSpeed:=0;
					m_dLastIntegral:=0;
					r_Integral_thistime:=0;
					r_el_offset_abs:=0;
					IF b_remote_on THEN
					i_receive_cmd:=i_receive_cmd+1;
					i_excute_cmd:=i_excute_cmd+1;
					last_command:='06';
					END_IF
				    str_Send:=F_RPL_1('',str_Send);
					b_commanding:=FALSE;
					b_sending:=TRUE;
			ELSE
				   	str_Send:=F_RPL_1('',str_Send);
					b_commanding:=FALSE;
					b_sending:=TRUE;
			END_IF;
(*<<<<<<<<<<<<<<<<<<<<<<<<<<<<<<<<<<<<<<ESTOP>>>>>>>>>>>>>>>>>>>>>>>>>>>>>>>>>>>>>>>>>>>>>>>*)
		ELSIF	fb_msg_receive.Key ='ESTOP'  AND b_remote_on=TRUE THEN
			b_power_Az :=FALSE;
			b_power_el:=FALSE;
			b_power_FI:=FALSE;
	     	str_Send:=F_RPL_1('',str_Send);
					b_commanding:=FALSE;
					b_sending:=TRUE;

(*<<<<<<<<<<<<<<<<<<<<<<<<<<<<<GOTO>>>>>>>>>>>>>>>>>>>>>>>>>>>>>>>>>>>>>>>>*)
		ELSIF fb_msg_receive.Key='GOTO'  THEN
			r_EL_current_when_goto_cmd:=r_pos_el;
			T_count_goto:=0.0;
			Pos_EL_Aim:=r_pos_el;
			r_goto_az_I:=STRING_TO_REAL(fb_msg_receive.P_value[1]);(*input value of GOTO*)
            r_goto_el_I:=STRING_TO_REAL(fb_msg_receive.P_value[2]);
            r_goto_FI_I:=STRING_TO_REAL(fb_msg_receive.P_value[3]);
				IF (-270.01<r_goto_az_I)AND(r_goto_az_I<270.01)AND(14.9<r_goto_el_I)AND(r_goto_el_I<=90)AND(-0.01<r_goto_FI_I)AND(r_goto_FI_I<180.01)THEN
					r_goto_az:=r_goto_az_I-r_pos_az_v;
					vel_move_az_1:=vel_move_az;
						acc_mov_az:=0.08;
						dcc_mov_az:=0.08;				
					b_scc_vel1_temp:=FALSE;
					b_start_adjust_vel:=FALSE;
					r_p0:=ML_Base.AxisData[11].rActualPosition_i;
					r_p1:=Encoder_to_motor(r_goto_el_I);
					r_p2:=Encoder_to_motor(r_p0);
					r_goto_el_abs:=Encoder_to_motor(r_goto_el_I);
					r_goto_el:=Encoder_to_motor(r_goto_el_I)-Encoder_to_motor(ML_Base.AxisData[11].rActualPosition_i);
					r_goto_FI:=r_goto_FI_I-r_pos_FI_v+90;
					b_first_pos_done:=FALSE;
					b_second_pos_done:=FALSE;
					b_3rd_pos_done:=FALSE;
					b_4th_pos_done:=FALSE;
					b_5th_pos_done:=FALSE;
					b_6th_pos_done:=FALSE;
					b_7th_pos_done:=FALSE;
					b_8th_pos_done:=FALSE;
					b_9th_pos_done:=FALSE;
					b_10th_pos_done:=FALSE;
					i_adjust_count:=0;
					adjust_delay:=FALSE;
					i_closeloop_count:=0;					
					b_SCC_STOP:=FALSE;
					b_scc_goto:=TRUE;
					b_start_goto_az_tcp:=TRUE;
					b_step_running_az:=1;
					b_step_running_el:=1;
					r_step_count_temp:=r_step_count_temp+1;
					b_in_positionMode:=TRUE;	
					IF b_remote_on THEN
					i_receive_cmd:=i_receive_cmd+1;
					i_excute_cmd:=i_excute_cmd+1;
					last_command:='02';
					END_IF
					str_Send:=F_RPL_1('',str_Send);
					b_commanding:=FALSE;
					b_sending:=TRUE;
				ELSE
					b_scc_goto:=FALSE;
					b_start_goto_az_tcp:=FALSE;
					str_Send:=F_RPL_1('',str_Send);
					b_commanding:=FALSE;
					b_sending:=TRUE;
				END_IF
(*<<<<<<<<<<<<<<<<<<<<<<<<<<<<<SETSPEED>>>>>>>>>>>>>>>>>>>>>>>>>>>>>>>>>>>>>>>>*)
		ELSIF fb_msg_receive.Key='SETSPEED'  THEN
			vel_move_az:=STRING_TO_REAL(fb_msg_receive.P_value[1])/6;
            vel_move_el:=STRING_TO_REAL(fb_msg_receive.P_value[2])/6;
            vel_move_FI:=STRING_TO_REAL(fb_msg_receive.P_value[3])/6;
			IF b_remote_on THEN
			i_receive_cmd:=i_receive_cmd+1;
			i_excute_cmd:=i_excute_cmd+1;
			last_command:='09';
			END_IF
				IF (vel_move_az>0.5)OR(vel_move_el>0.167)OR(vel_move_FI>0.334)THEN
					IF vel_move_az>0.5 THEN
						vel_move_az:=0.5;
					END_IF
					IF vel_move_el>0.167 THEN
						vel_move_el:=0.167;
					END_IF
					IF vel_move_FI>0.334 THEN
						vel_move_FI:=0.334;
					END_IF	
								
					str_Send:=F_RPL_1('',str_Send);
					b_commanding:=FALSE;
					b_sending:=TRUE;
				ELSE
					str_Send:=F_RPL_1('',str_Send);
					b_commanding:=FALSE;
					b_sending:=TRUE;
				END_IF				
				
				
(*<<<<<<<<<<<<<<<<<<<<<<<<<<<<<VEL>>>>>>>>>>>>>>>>>>>>>>>>>>>>>>>>>>>>>>>>*)
		ELSIF fb_msg_receive.Key='VEL' THEN
			b_scc_goto:=FALSE;
			b_scc_vel:=FALSE;
			b_SCC_STOP:=FALSE;
			b_track_on:=FALSE;
			V_command_EL:=0;
			V_LastSpeed:=0;
			V_LastOutput:=0;
			dIntegralSpeed:= 0;	
			b_start_cyclicvel:=FALSE;
			b_write_el_vel:=FALSE;
			b_start_adjust_vel_temp:=FALSE;
			b_start_adjust_vel:=FALSE;
			r_vel_az:=STRING_TO_REAL(fb_msg_receive.P_value[1])/6;
            r_vel_el:=STRING_TO_REAL(fb_msg_receive.P_value[2])/6;
			r_command_vel:=r_vel_el*6;
            r_vel_FI:=STRING_TO_REAL(fb_msg_receive.P_value[3])/6;
			IF b_remote_on_run=FALSE THEN
					str_Send:=F_RPL_1('',str_Send);
					b_commanding:=FALSE;
					b_sending:=TRUE;
			ELSE
				IF (-0.51<r_vel_az)AND(r_vel_az<0.51)AND(-0.17<r_vel_el)AND(r_vel_el<0.17)AND(-0.334<r_vel_FI)AND(r_vel_FI<0.334)THEN
					IF r_pos_az_v>265 AND r_vel_az>0.083 THEN
						r_vel_az:=0.083;
					END_IF
					
					IF r_pos_az_v<-265 AND r_vel_az<-0.083 THEN
						r_vel_az:=-0.083;
					END_IF
					
					IF r_pos_el_v>88 AND r_vel_el>0.1 THEN
						r_vel_el:=0.05;
					END_IF
					
					IF r_pos_el_v<20 AND r_vel_el<-0.1 THEN
						r_vel_el:=-0.05;
					END_IF

					IF r_pos_FI_v>265 AND r_vel_FI>0.083 THEN
						r_vel_FI:=0.083;
					END_IF
					
					IF r_pos_FI_v<95 AND r_vel_FI<-0.083 THEN
						r_vel_FI:=-0.083;
					END_IF
					r_vel_el:=r_vel_el*11976;//*7.5;
//					r_vel_el:=r_vel_el*12100;//*7.5;
					b_scc_vel:=TRUE;
					str_Send:=F_RPL_1('',str_Send);
					b_commanding:=FALSE;
					b_sending:=TRUE;
				ELSE
					b_scc_vel:=FALSE;
				    str_Send:=F_RPL_1('',str_Send);
					b_commanding:=FALSE;
					b_sending:=TRUE;
				END_IF
			END_IF			
			
(*<<<<<<<<<<<<<<<<<<<<<<<<<<<<<<<<<<<<<<POWER>>>>>>>>>>>>>>>>>>>>>>>>>>>>>>>>>>>>>>>>>>>>>>>*)
		ELSIF fb_msg_receive.Key ='PWR'  THEN
				lockstand:=TRUE;
			IF fb_msg_receive.P_value[1]='ON' THEN
				b_power_on:=FALSE;
				IF axisdata[1].Axis_InAb = 0 THEN
				b_Scc_PWR_on:=FALSE;
				b_Scc_PWR_on:=TRUE;
				b_Scc_PWR_off:=FALSE;
				END_IF;
					str_Send:=F_RPL_1('',str_Send);
					b_commanding:=FALSE;
					b_sending:=TRUE;
			ELSIF fb_msg_receive.P_value[1]='OFF' THEN
				IF b_track_on=FALSE THEN
					b_Scc_PWR_on:=FALSE;
					b_Scc_PWR_off:=TRUE;
					b_scc_goto:=FALSE;
					b_active_AZ:=FALSE;
					b_active_EL:=FALSE;
					b_scc_vel:=FALSE;
					b_active_FI:=FALSE;
					b_goto_Az_done:=FALSE;
					b_goto_EL_done:=FALSE;
					b_goto_FI_done:=FALSE;
					b_SCC_STOP:=FALSE;
					b_stop_act_az:=FALSE;
					b_stop_act_el:=FALSE;
					b_stop_act_FI:=FALSE;
					b_stop1_done:=FALSE;
					b_stop3_done:=FALSE;
					b_stop5_done:=FALSE;
					b_scc_maintain:=FALSE;
					b_scc_stow:=FALSE;
					b_write_az:=FALSE;
					b_write_el:=FALSE;
					b_write_FI:=FALSE;
					b_write_az_done:=FALSE;
					b_write_el_done:=FALSE;
					b_write_FI_done:=FALSE;
					b_open_channel_az:=FALSE;
					b_open_channel_el:=FALSE;
					b_open_channel_FI:=FALSE;
					b_open_channel_az_done:=FALSE;
					b_open_channel_el_done:=FALSE;
					b_open_channel_FI_done:=FALSE;
					b_move_0_done:=FALSE;
					b_move_20_done:=FALSE;
					b_lock_off:=FALSE;
					str_Send:=F_RPL_1('',str_Send);
					b_commanding:=FALSE;
					b_sending:=TRUE;
				ELSE
					str_Send:=F_RPL_1('',str_Send);
					b_commanding:=FALSE;
					b_sending:=TRUE;
				END_IF
			ELSE
				   	str_Send:=F_RPL_1('',str_Send);
					b_commanding:=FALSE;
					b_sending:=TRUE;
			END_IF
(*<<<<<<<<<<<<<<<<<<<<<<<<<<<<<<<<<<<<<<STOP>>>>>>>>>>>>>>>>>>>>>>>>>>>>>>>>>>>>>>>>>>>>>>>*)
		ELSIF fb_msg_receive.Key ='STOP' THEN
		
				IF b_track_on=TRUE THEN
					b_stop_TOA:=TRUE;				
				ELSE
					b_on_track_mode:=FALSE;
					b_track_on_first:=FALSE;
					i_start:=1;
					i_end:=1;
					b_Track_Pause:=FALSE;
					track_table[1].TAIoffset:=0;
					FOR i_count:=1 TO i_total BY 1 DO
					track_table[i_count].TAIoffset:=0;
					track_table[i_count].Azimuth:= 0;
					track_table[i_count].Elevation:=0;
					//track_table[i_count].FeedIndexer:=0;
					//track_table[i_count].Elevation_ori:=0;
					END_FOR;
					(*track_table[1].MJD:=0;
					FOR i_count:=1 TO i_total BY 1 DO
					track_table[i_count].MJD:=0;
					track_table[i_count].Azimuth:= 0;
					track_table[i_count].Elevation:=0;
					track_table[i_count].FeedIndexer:=0;
					track_table[i_count].Elevation_ori:=0;
					END_FOR;*)
					b_SCC_STOP:=TRUE;
					V_LastSpeed:=0;
					V_LastOutput:=0;
					dIntegralSpeed:= 0;	
					V_command_EL:=0;
					b_start_cyclicvel:=FALSE;
					b_write_el_vel:=FALSE;	
					b_Track_Pause:=FALSE;				
				END_IF
				b_SCC_goto:=FALSE;
				IF b_remote_on THEN
				i_receive_cmd:=i_receive_cmd+1;
				i_excute_cmd:=i_excute_cmd+1;
				last_command:='01';
				END_IF
				str_Send:=F_RPL_1('',str_Send);
				b_commanding:=FALSE;
				b_sending:=TRUE;
(*<<<<<<<<<<<<<<<<<<<<<<<<<<<<<<<<<<<<<<STOW>>>>>>>>>>>>>>>>>>>>>>>>>>>>>>>>>>>>>>>>>>>>>>>*)
		ELSIF fb_msg_receive.Key ='STOW' THEN
			b_scc_Unlock:=FALSE;
			IF b_PID_in_el=TRUE THEN
				b_scc_maintain:=FALSE;
				b_scc_stow:=TRUE;
					str_Send:=F_RPL_1('',str_Send);
					b_commanding:=FALSE;
					b_sending:=TRUE;
			ELSE
					str_Send:=F_RPL_1('',str_Send);
					b_commanding:=FALSE;
					b_sending:=TRUE;
			END_IF
(*<<<<<<<<<<<<<<<<<<<<<<<<<<<<<<<<<<<<<<MAINTAIN>>>>>>>>>>>>>>>>>>>>>>>>>>>>>>>>>>>>>>>>>>>>>>>*)
		ELSIF fb_msg_receive.Key ='MAINTAIN'  THEN
		
					b_permit_new_file:=TRUE;		
					str_Send:=F_RPL_1('',str_Send);
					b_commanding:=FALSE;
					b_sending:=TRUE;
			
(*<<<<<<<<<<<<<<<<<<<<<<<<<<<<<<<<<<<<<<HOME>>>>>>>>>>>>>>>>>>>>>>>>>>>>>>>>>>>>>>>>>>>>>>>*)
		ELSIF fb_msg_receive.Key ='HOME' THEN
		
					b_off_write:=FALSE;	
				    b_SCC_enable_off:=FALSE;
					IF b_remote_on THEN	
					i_receive_cmd:=i_receive_cmd+1;
					i_excute_cmd:=i_excute_cmd+1;
					last_command:='08';
					END_IF
			IF b_encoder_ok_az = FALSE THEN 
				B_encoder_home_d1:=TRUE;  
			END_IF
			
			IF b_encoder_ok_FI = FALSE THEN 
				B_encoder_home_d5:=TRUE;
			END_IF			
					str_Send:=F_RPL_1('',str_Send);
					b_commanding:=FALSE;
					b_sending:=TRUE;
				
(*<<<<<<<<<<<<<<<<<<<<<<<<<<<<<<<<<<<<<<unlock>>>>>>>>>>>>>>>>>>>>>>>>>>>>>>>>>>>>>>>>>>>>>>>*)
		ELSIF fb_msg_receive.Key ='UNLOCK' AND b_remote_on=TRUE THEN
			IF b_stow_pin_limit_unlock=TRUE  THEN
				b_scc_stow:=FALSE;
				b_scc_maintain:=FALSE;
				b_scc_Unlock:=TRUE;
					str_Send:=F_RPL_1('',str_Send);
					b_commanding:=FALSE;
					b_sending:=TRUE;
			ELSE
					str_Send:=F_RPL_1('',str_Send);
					b_commanding:=FALSE;
					b_sending:=TRUE;
			END_IF
(*<<<<<<<<<<<<<<<<<<<<<<<<<<<<<TRACK>>>>>>>>>>>>>>>>>>>>>>>>>>>>>>>>>>>>>>>>>>>>>>>>>>>>>>>*)
		ELSIF fb_msg_receive.Key='TRACK'  THEN
				b_scc_goto:=FALSE;
			IF fb_msg_receive.P_value[1]='ON' THEN
				IF b_remote_on_run=TRUE  THEN
					IF i_end<>i_START THEN
						b_track_on:=TRUE;
						b_stop_TOA:=FALSE;
						b_not_track:=FALSE;
						b_track_on_first:=TRUE;
						b_on_track_mode:=TRUE;
					b_Track_Pause:=FALSE;
					IF b_remote_on THEN
					i_receive_cmd:=i_receive_cmd+1;
					i_excute_cmd:=i_excute_cmd+1;
					last_command:='03';
					END_IF
					str_Send:=F_RPL_1('',str_Send);
					b_commanding:=FALSE;
					b_sending:=TRUE;
					ELSE
					str_Send:=F_RPL_1('',str_Send);
					b_commanding:=FALSE;
					b_sending:=TRUE;
					END_IF
				ELSE
					str_Send:=F_RPL_1('',str_Send);
					b_commanding:=FALSE;
					b_sending:=TRUE;
				END_IF
			ELSIF fb_msg_receive.P_value[1]='OFF' THEN
				
					b_track_on:=FALSE;
					b_on_track_mode:=FALSE;
					b_track_on_first:=FALSE;
					i_start:=1;
					i_end:=1;
					b_Track_Pause:=FALSE;
					track_table[1].TAIoffset:=0;
					FOR i_count:=1 TO i_total BY 1 DO
					track_table[i_count].TAIoffset:=0;
					track_table[i_count].Azimuth:= 0;
					track_table[i_count].Elevation:=0;
					//track_table[i_count].FeedIndexer:=0;
					//track_table[i_count].Elevation_ori:=0;
					END_FOR;
				(*	track_table[1].MJD:=0;
					FOR i_count:=1 TO i_total BY 1 DO
					track_table[i_count].MJD:=0;
					track_table[i_count].Azimuth:= 0;
					track_table[i_count].Elevation:=0;
					track_table[i_count].FeedIndexer:=0;
					track_table[i_count].Elevation_ori:=0;
					END_FOR; *)
//					b_SCC_STOP:=TRUE;
					b_Track_Pause:=FALSE;				
					b_SCC_goto:=FALSE;
			
(*					
				IF i_start<>i_end THEN
				
					i_pause_temp:=i_start;
					t_difference:=(entry_buffer1[F_I_number(i_start)].MJD-entry_buffer1[F_I_number(i_start-1)].MJD)*86400;
					r_a0:=entry_buffer1[F_I_number(i_start)].Azimuth-entry_buffer1[F_I_number(i_start-1)].Azimuth;
					v_a0:=r_a0/t_difference;
					a_a0:=-v_a0/3;
					i_stop:=ABS(REAL_TO_INT(2.0/t_difference));
					i_stop_1:=ABS(REAL_TO_INT(5/t_difference));

			
					r_az_pause_pos1:=r_pos_az_v + v_a0*0.5 + 0.5*a_a0*0.5*0.5;
					r_az_pause_pos2:=r_pos_az_v + v_a0*1 + 0.5*a_a0*1*1;
					r_az_pause_pos3:=r_pos_az_v + v_a0*1.5 + 0.5*a_a0*1.5*1.5;
					r_az_pause_pos4:=r_pos_az_v + v_a0*2 + 0.5*a_a0*2*2;
					r_az_pause_pos5:=r_pos_az_v + v_a0*2.5 + 0.5*a_a0*2.5*2.5;
					r_az_pause_pos6:=r_pos_az_v + v_a0*3 + 0.5*a_a0*3*3;
					r_az_pause_pos7:=r_pos_az_v + v_a0*3 + 0.5*a_a0*3*3;
					
					entry_buffer1[F_I_number(i_start+1)].Azimuth:=r_az_pause_pos1;
					entry_buffer1[F_I_number(i_start+2)].Azimuth:=r_az_pause_pos2;
					entry_buffer1[F_I_number(i_start+3)].Azimuth:=r_az_pause_pos3;
					entry_buffer1[F_I_number(i_start+4)].Azimuth:=r_az_pause_pos4;
					entry_buffer1[F_I_number(i_start+5)].Azimuth:=r_az_pause_pos5;
					entry_buffer1[F_I_number(i_start+6)].Azimuth:=r_az_pause_pos6;
					entry_buffer1[F_I_number(i_start+7)].Azimuth:=r_az_pause_pos7;
					entry_buffer1[F_I_number(i_start+8)].Azimuth:=r_az_pause_pos7;
					entry_buffer1[F_I_number(i_start+9)].Azimuth:=r_az_pause_pos7;
					entry_buffer1[F_I_number(i_start+10)].Azimuth:=r_az_pause_pos7;
										
					entry_buffer1[F_I_number(i_start+1)].MJD:=lr_MJD_current+0.0000058;
					entry_buffer1[F_I_number(i_start+2)].MJD:=lr_MJD_current+0.0000058*2;
					entry_buffer1[F_I_number(i_start+3)].MJD:=lr_MJD_current+0.0000058*3;
					entry_buffer1[F_I_number(i_start+4)].MJD:=lr_MJD_current+0.0000058*4;
					entry_buffer1[F_I_number(i_start+5)].MJD:=lr_MJD_current+0.0000058*5;
					entry_buffer1[F_I_number(i_start+6)].MJD:=lr_MJD_current+0.0000058*6;	
					entry_buffer1[F_I_number(i_start+7)].MJD:=lr_MJD_current+0.0000058*7;	
					entry_buffer1[F_I_number(i_start+8)].MJD:=lr_MJD_current+0.0000058*8;	
					entry_buffer1[F_I_number(i_start+9)].MJD:=lr_MJD_current+0.0000058*9;	
					entry_buffer1[F_I_number(i_start+10)].MJD:=lr_MJD_current+0.0000058*10;	
			END_IF			
										
                    IF b_on_track_mode THEN 
						b_Track_Pause:=TRUE;
					END_IF
*)
					b_track_on_first:=FALSE;
						
					str_Send:=F_RPL_1('',str_Send);
					b_commanding:=FALSE;
					b_sending:=TRUE;
			END_IF
(*<<<<<<<<<<<<<<<<<<<<<<<<<<<<<TRKVAL>>>>>>>>>>>>>>>>>>>>>>>>>>>>>>>>>>>>>>>>>>>>>>>>>>>>>>>*)
		ELSIF fb_msg_receive.Key='TRKVAL'  THEN
			IF fb_msg_receive.P_value[1]='OFF' THEN
				i_start:=1;
				i_end:=1;
				b_on_track_mode:=FALSE;
				b_track_on_first:=FALSE;
				b_track_on:=FALSE;
				b_Track_Pause:=FALSE;
				track_table[1].TAIoffset:=0;
				FOR i_count:=1 TO i_total BY 1 DO
					track_table[i_count].TAIoffset:=0;
					track_table[i_count].Azimuth:= 0;
					track_table[i_count].Elevation:=0;
					//track_table[i_count].FeedIndexer:=0;
				END_FOR;
			(*	track_table[1].MJD:=0;
				FOR i_count:=1 TO i_total BY 1 DO
					track_table[i_count].MJD:=0;
					track_table[i_count].Azimuth:= 0;
					track_table[i_count].Elevation:=0;
					track_table[i_count].FeedIndexer:=0;
				END_FOR; *)
					str_Send:=F_RPL_1('',str_Send);
					b_commanding:=FALSE;
					b_sending:=TRUE;
			ELSE
			fb_Trkval(
				str_MJD:=fb_msg_receive.P_value[1],
				str_Azimuth:=fb_msg_receive.P_value[2],
				str_Elevation:=fb_msg_receive.P_value[3],
	        	str_FeedIndexer:=fb_msg_receive.P_value[4]);
				
				b_not_track:=false;	
				b_permit_new_file:=FALSE;
				str_Send:=F_RPL_1('',str_Send);
					b_commanding:=FALSE;
					b_sending:=TRUE;
			END_IF;
(*<<<<<<<<<<<<<<<<<<<<<<<<<<<<<UPDATE of NTP>>>>>>>>>>>>>>>>>>>>>>>>>>>>>>>>>>>>>>>>>>>>>>>>>>>>>>>*)
		ELSIF fb_msg_receive.Key='SNTP' THEN
			IF b_track_on=FALSE THEN
				b_NTP_update_start:=TRUE;
					str_Send:=F_RPL_1('',str_Send);
					b_commanding:=FALSE;
					b_sending:=TRUE;
			ELSE
					str_Send:=F_RPL_1('',str_Send);
					b_commanding:=FALSE;
					b_sending:=TRUE;
			END_IF
(*<<<<<<<<<<<<<<<<<<<<<<<<<<<<<GSTAT>>>>>>>>>>>>>>>>>>>>>>>>>>>>>>>>>>>>>>>>>>>>>>>>>>>>>>>*)
		ELSIF fb_msg_receive.Key='GSTAT' THEN


      		      	str_Send:=F_RPL_1('',str_Send);
					b_commanding:=FALSE;
					b_sending:=TRUE;
(*<<<<<<<<<<<<<<<<<<<<<<<<<<<<<<<<<<<<<<K1STAT>>>>>>>>>>>>>>>>>>>>>>>>>>>>>>>>>>>>>>>>>>>>>>>*)
		ELSIF fb_msg_receive.Key ='K1STAT' THEN
			str_Send:='OK - CECT54_12m_V1.1 006-336-918 -179 359 15 90.1 -179 179 90 0 0 0';
					b_commanding:=FALSE;
					b_sending:=TRUE;
(*<<<<<<<<<<<<<<<<<<<<<<<<<<<<<<<<<<<<<<K2STAT>>>>>>>>>>>>>>>>>>>>>>>>>>>>>>>>>>>>>>>>>>>>>>>*)
		ELSIF fb_msg_receive.Key ='K2STAT' THEN
				str_Send:=F_RPL_1('',str_Send);
					b_commanding:=FALSE;
					b_sending:=TRUE;
(*<<<<<<<<<<<<<<<<<<<<<<<<<<<<<<<<<<<<<<K3STAT>>>>>>>>>>>>>>>>>>>>>>>>>>>>>>>>>>>>>>>>>>>>>>>*)
		ELSIF fb_msg_receive.Key ='K3STAT' THEN
			status_K3.0:=b_estop_dr;
			status_K3.1:=b_estop_az;
			status_K3.2:=b_estop_el;
			status_K3.3:=b_estop_FI;
			status_K3.4:=b_estop_mc;
			str_Send:=CONCAT('OK - ',DWORD_TO_STRING(status_K3));
					b_commanding:=FALSE;
					b_sending:=TRUE;
					
(*<<<<<<<<<<<<<<<<<<<<<<<<<<<<<<<<<<<<<<LOCKSTANDBY>>>>>>>>>>>>>>>>>>>>>>>>>>>>>>>>>>>>>>>>>>>>>>>*)
		ELSIF	fb_msg_receive.Key ='LOCKSTANDBY' THEN
				i_counter_1s:=0;
				b_stow:=FALSE;
				b_power_on:=FALSE;
				b_Scc_PWR_on:=FALSE;
				lockstand:=TRUE;
				b_track_on:=FALSE;	
				b_SCC_enable_on:=FALSE;
				b_SCC_enable_off:=FALSE;	
				b_off_write:=FALSE;	
			  	str_Send:=F_RPL_1('',str_Send);
					b_commanding:=FALSE;
					b_sending:=TRUE;			
(***********************OFFSET*************************)
    	 ELSIF fb_msg_receive.Key='OFFSET' THEN
			i_counter_1s:=0;
			r_offset_az_I:=STRING_TO_REAL(fb_msg_receive.P_value[1]);
            r_offset_el_I:=STRING_TO_REAL(fb_msg_receive.P_value[2]);
			
			IF b_track_on  THEN
				b_offset:=TRUE;
				b_test_offset_start:=TRUE;
				str_Send:=F_RPL_1('',str_Send);;
			ELSE
				b_offset:=FALSE;
				b_test_offset_start:=FALSE;
				str_Send:=F_RPL_1('',str_Send);
			END_IF
					b_commanding:=FALSE;
					b_sending:=TRUE;	
(*新加入的累计偏置，一次只能识别加减一次*)
(*				r_offset_az:=r_offset_az+r_offset_az_I;
				r_offset_el:=r_offset_el+r_offset_el_I;
*)
				r_offset_az:=r_offset_az_I-r_offset_az_old;
				r_offset_el:=r_offset_el_I-r_offset_el_old;
//				r_offset_el_program:=r_offset_el_I;
			IF r_offset_az_I=0 AND r_offset_el_I=0 THEN
				r_offset_az:=-r_offset_az_old;
				r_offset_el:=-r_offset_el_old;
				b_offset_running:=TRUE;
				r_offset_count_temp:=r_offset_count_temp+1;
			END_IF;					
(*<<<<<<<<<<<<<<<<<<<<<<<<<<<<<<<<<<<<<<K4STAT>>>>>>>>>>>>>>>>>>>>>>>>>>>>>>>>>>>>>>>>>>>>>>>*)
		ELSIF fb_msg_receive.Key ='K4STAT' THEN
				str_Send:=F_RPL_1('',str_Send);
					b_commanding:=FALSE;
					b_sending:=TRUE;
(*<<<<<<<<<<<<<<<<<<<<<<<<<<<<<<<<<<<<<K5STAT>>>>>>>>>>>>>>>>>>>>>>>>>>>>>>>>>>>>>>>>>>>>>>>>*)
		ELSIF fb_msg_receive.Key ='K5STAT' THEN
				str_Send:=F_RPL_1('',str_Send);
					b_commanding:=FALSE;
					b_sending:=TRUE;
(*<<<<<<<<<<<<<<<<<<<<<<<<<<<<<<<<<<<<<<VERSION>>>>>>>>>>>>>>>>>>>>>>>>>>>>>>>>>>>>>>>>>>>>>>>*)
		ELSIF fb_msg_receive.Key ='VERSION' THEN
			str_Send:=CONCAT('VERSION=V1.1',' CETC54 27 JUL 2015 Alex');
				
					b_commanding:=FALSE;
					b_sending:=TRUE;
(*<<<<<<<<<<<<<<<<<<<<<<<<<<<<<<<<<<<<<<TSTAT>>>>>>>>>>>>>>>>>>>>>>>>>>>>>>>>>>>>>>>>>>>>>>>*)
		ELSIF fb_msg_receive.Key='TSTAT' THEN
			str_Send:=CONCAT('OK -',CONCAT(' ',INT_TO_STRING(i_num_stack_left)));
 			str_Send:=CONCAT(str_Send,CONCAT(' ',REAL_TO_STRING(r_track_error[1])));
			str_Send:=CONCAT(str_Send,CONCAT(' ',REAL_TO_STRING(r_track_error[2])));
			str_Send:=CONCAT(str_Send,CONCAT(' ',REAL_TO_STRING(r_track_error[3])));
					b_commanding:=FALSE;
					b_sending:=TRUE;
		ELSE
			IF b_remote_on=FALSE THEN
					str_Send:=F_RPL_1('',str_Send);
					b_commanding:=FALSE;
					b_sending:=TRUE;
			ELSE
					str_Send:=F_RPL_1('',str_Send);
					b_commanding:=FALSE;
					b_sending:=TRUE;
			END_IF
		END_IF;
	END_IF;
	

